(* HMI Lights Control *) //-----------------------------------------------------------------------------------------------
GVL_IO.gRelayOutputs.bSampleRecoveryLight 		:= GVL_HMI.bLightsToggleButton;
GVL_IO.gRelayOutputs.bStageCollectionLeftLight 	:= GVL_HMI.bLightsToggleButton;
GVL_IO.gRelayOutputs.bStageCollectionRightLight := GVL_HMI.bLightsToggleButton;

(* <Linear Pumps Old Position> ----------------------------------------------------------------------------------------- *)
// display linear pumps old position saved on persistent memory when in Calibration Mode
IF GVL_HMI.eMachineMode = E_MachineMode.CALIBRATION THEN
	FOR i := 1 TO 10 DO
		IF GVL_Motion.aPumps[i].Linear.iHomed THEN
			GVL_HMI.aCalibLinearPumps[1].rNewPosition := GVL_Motion.aPumps[i].Linear.rActualPos;
		END_IF
	END_FOR
END_IF

(* <Pump Factor Showing> ----------------------------------------------------------------------------------------------- *)
(*IF GVL_HMI.eMachineMode = E_MachineMode.CALIBRATION THEN
	FOR i := 1 TO 10 DO
		GVL_HMI.aCalPumpResults[i].rPumpFactor := GVL_Motion.aPumps[i].Rotary.rPumpFactorFromCalBox;
	END_FOR
END_IF
*)

(* <Safety Controls> ----------------------------------------------------------------------------------------------------*)
ton500ms(IN := NOT ton500ms.Q, PT := T#500MS);

IF ton500ms.Q THEN ACT_IOControls(); END_IF

//Calibration Box presence
GVL_HMI.bHMICalibrationBox := GVL_IO.gDigInputs.bCalibrationBoxPresent;

//Valves Angle
GVL_HMI.HMIAnimation.aValveAngle[1]	:= GVL_Motion.aValves[1].rActualPosition / 60;
GVL_HMI.HMIAnimation.aValveAngle[2]	:= GVL_Motion.aValves[2].rActualPosition / 60;;
GVL_HMI.HMIAnimation.aValveAngle[3]	:= GVL_Motion.aValves[3].rActualPosition / 60;;
GVL_HMI.HMIAnimation.aValveAngle[4]	:= GVL_Motion.aValves[4].rActualPosition / 60;;
GVL_HMI.HMIAnimation.aValveAngle[5]	:= GVL_Motion.aValves[5].rActualPosition / 60;;

//Pumps status Running or busy
IF GVL_HMI.eMachineMode = E_MachineMode.MANUAL THEN
	FOR i := 1 TO 10 DO
		aPumpStatus[i] := GVL_Motion.aPumpsRotary[i].GetStatus();
		GVL_HMI.aManualPumpsCmd[i].bBusy := NOT GVL_Motion.aPumps[i].Rotary.iNotMoving; //aPumpStatus[i].bBusy;
	END_FOR
END_IF

//Check if there is at least one pump running
GVL_Motion.bAnyPumpRunning := FALSE;
FOR i := 1 TO 10 DO
	IF GVL_HMI.aManualPumpsCmd[i].bBusy THEN
		GVL_Motion.bAnyPumpRunning := TRUE;
		EXIT;
	END_IF
END_FOR


//Pumps Animation | Calibration Screen
IF GVL_HMI.eMachineMode = E_MachineMode.CALIBRATION THEN
	ACT_CalibrationArrows();
END_IF

//Scan period for hmi refresh
//IF GVL_HMI.eMachineMode <> E_MachineMode.CALIBRATION AND GVL_HMI.eMachineMode <> E_MachineMode.MANUAL THEN
	fbHMIScan(bEnable := GVL_HMI.bHomeScreenLoaded, tPeriod := T#500MS);
	GVL_HMI.bMachineModeScan := fbHMIScan.bBlink;
//ELSE
//	GVL_HMI.bMachineModeScan := FALSE;
//END_IF

// Home Rotary Pumps direction cover
IF GVL_HMI.bHomeScreenLoaded THEN
	FOR i := 1 TO 10 DO
		GVL_HMI.HMIAnimation.bPumpPositiveDirection[i] := GVL_Motion.aPumps[i].Rotary.bPositiveDirection;
		GVL_HMI.HMIAnimation.bPumpNegativeDirection[i] := GVL_Motion.aPumps[i].Rotary.bNegativeDirection;
	END_FOR	
END_IF

//Doors hide/visible 
GVL_HMI.HMIAnimation.bHMIDoorOpen[1] := NOT GVL_Safety.SafetyInputs.bStageCollectLeftDoorFdbk;
GVL_HMI.HMIAnimation.bHMIDoorOpen[2] := NOT GVL_Safety.SafetyInputs.bStageCollectRightDoorFdbk;
GVL_HMI.HMIAnimation.bHMIDoorOpen[3] := NOT GVL_Safety.SafetyInputs.bSampleRecoveryDoorFdbk;
GVL_HMI.HMIAnimation.bHMIDoorOpen[4] := GVL_IO.gDigInputs.bAccessDoor4InterlockFdbk;
GVL_HMI.HMIAnimation.bHMIDoorOpen[5] := GVL_IO.gDigInputs.bAccessDoor5InterlockFdbk;
GVL_HMI.HMIAnimation.bHMIDoorOpen[6] := GVL_IO.gDigInputs.bAccessDoor6InterlockFdbk;

//Doors open blinking red alert
fbBlinkDoor[1](bEnable := NOT GVL_Safety.SafetyInputs.bStageCollectLeftDoorFdbk, tPeriod := T#1S);
GVL_HMI.HMIAnimation.bHMIDoorBlink[1] := fbBlinkDoor[1].bBlink;

fbBlinkDoor[2](bEnable := NOT GVL_Safety.SafetyInputs.bStageCollectRightDoorFdbk, tPeriod := T#1S);
GVL_HMI.HMIAnimation.bHMIDoorBlink[2] := fbBlinkDoor[2].bBlink;

fbBlinkDoor[3](bEnable := NOT GVL_Safety.SafetyInputs.bSampleRecoveryDoorFdbk, tPeriod := T#1S);
GVL_HMI.HMIAnimation.bHMIDoorBlink[3] := fbBlinkDoor[3].bBlink;

fbBlinkDoor[4](bEnable := GVL_IO.gDigInputs.bAccessDoor4InterlockFdbk, tPeriod := T#1S);
GVL_HMI.HMIAnimation.bHMIDoorBlink[4] := fbBlinkDoor[4].bBlink;

fbBlinkDoor[5](bEnable := GVL_IO.gDigInputs.bAccessDoor5InterlockFdbk, tPeriod := T#1S);
GVL_HMI.HMIAnimation.bHMIDoorBlink[5] := fbBlinkDoor[5].bBlink;

fbBlinkDoor[6](bEnable := GVL_IO.gDigInputs.bAccessDoor6InterlockFdbk, tPeriod := T#1S);
GVL_HMI.HMIAnimation.bHMIDoorBlink[6] := fbBlinkDoor[6].bBlink;


(* <\Controls Animation> *********************************************************************************************** *)

(* <Icons Animation> *************************************************************************************************** *)
IF NOT bFirstIconSet THEN
	GVL_HMI.HMIAnimation.eIconStateSafety   := E_IconState.Waiting;
	GVL_HMI.HMIAnimation.eIconStateAirFlow  := E_IconState.Waiting;
	GVL_HMI.HMIAnimation.eIconStateSealing 	:= E_IconState.Waiting;
	GVL_HMI.HMIAnimation.eIconStateHardware := E_IconState.Waiting;
	GVL_HMI.HMIAnimation.eIconStatePrime 	:= E_IconState.Waiting;
	GVL_HMI.HMIAnimation.eIconStateLeakTest := E_IconState.Waiting;
	GVL_HMI.HMIAnimation.eIconStateRecovery := E_IconState.Waiting;
	GVL_HMI.HMIAnimation.eIconStateWashing  := E_IconState.Waiting;
	GVL_HMI.HMIAnimation.eIconStateDry 		:= E_IconState.Waiting;
	bFirstIconSet := TRUE;
END_IF

IF GVL_HMI.eMachineMode = E_MachineMode.IMEDIATE_FAULT THEN
	GVL_HMI.HMIAnimation.eIconStateSafety   := E_IconState.Waiting;
	GVL_HMI.HMIAnimation.eIconStateAirFlow  := E_IconState.Waiting;
	GVL_HMI.HMIAnimation.eIconStateSealing  := E_IconState.Waiting;
	GVL_HMI.HMIAnimation.eIconStateHardware := E_IconState.Waiting;
	GVL_HMI.HMIAnimation.eIconStatePrime  	:= E_IconState.Waiting;
	GVL_HMI.HMIAnimation.eIconStateLeakTest := E_IconState.Waiting;
	GVL_HMI.HMIAnimation.eIconStateRecovery := E_IconState.Waiting;
	GVL_HMI.HMIAnimation.eIconStateWashing  := E_IconState.Waiting;
	GVL_HMI.HMIAnimation.eIconStateDry 	    := E_IconState.Waiting;
ELSE
	GVL_HMI.HMIAnimation.eIconStateSafety := E_IconState.Completed;
END_IF

IF GVL_HMI.eMachineMode = E_MachineMode.STOPPED THEN
	GVL_HMI.HMIAnimation.eIconStateSafety   := E_IconState.Waiting;
	GVL_HMI.HMIAnimation.eIconStateAirFlow  := E_IconState.Waiting;
	GVL_HMI.HMIAnimation.eIconStateSealing 	:= E_IconState.Waiting;
	GVL_HMI.HMIAnimation.eIconStateHardware := E_IconState.Waiting;
	GVL_HMI.HMIAnimation.eIconStatePrime 	:= E_IconState.Waiting;
	GVL_HMI.HMIAnimation.eIconStateLeakTest := E_IconState.Waiting;
	GVL_HMI.HMIAnimation.eIconStateRecovery := E_IconState.Waiting;
	GVL_HMI.HMIAnimation.eIconStateWashing  := E_IconState.Waiting;
	GVL_HMI.HMIAnimation.eIconStateDry 	    := E_IconState.Waiting;
END_IF

(* <\Icons Animation> *************************************************************************************************** *)

(* <Machine Settings> ************************************************************************************************** *)
IF GVL_HMI.bSaveParametersBt THEN // Save Settings button from HMI
	GVL_Settings.stMachineParam	 		:= GVL_HMI.HMIParameters; 		 // Motion Settings
	GVL_Settings.stCalibParameters 		:= GVL_HMI.stHMICalibParameters; // Calibration Settings
	GVL_Settings.stPumpParameters 		:= GVL_HMI.stHMIPumpParameters;	 // Pump Settings
	GVL_Settings.stLeakTestParameters 	:= GVL_HMI.stLeakTestParameters; // Leak Test Settings
	GVL_Settings.sLastSysSettingsChangedBy 	:= GVL_HMI.sUserNameEventTriggered;
	GVL_Settings.sLastSysSettingsChangedOn 	:= GVL_HMI.sDateAndTimeEventTriggered;
	GVL_Settings.sysRevNumber 				:= GVL_Settings.sysRevNumber + 1;
	DB_Query.state:= E_DB_QUERY_STATE.INSERT_SYS_PARAMETERS;	// DB writing
	GVL_HMI.bSaveParametersBt 	:= FALSE;
	GVL_HMI.bSaveParametersDone := TRUE;
END_IF

IF GVL_HMI.bReloadHMIParameters OR (GVL_HMI.eMachineMode = E_MachineMode.CALIBRATION) THEN
	GVL_HMI.HMIParameters := GVL_Settings.stMachineParam;				 // Motion Settings
	GVL_HMI.stHMICalibParameters := GVL_Settings.stCalibParameters; 	 // Calibration Settings
	GVL_HMI.stHMIPumpParameters  := GVL_Settings.stPumpParameters; 		 // Pump Settings
	GVL_HMI.stLeakTestParameters := GVL_Settings.stLeakTestParameters; 	 // Leak Test Settings
	GVL_HMI.bReloadHMIParameters := FALSE;
END_IF

// Solvents Section [Database insert done via HMI]
PRG_SaveSolvents();
(*
IF GVL_HMI.bSaveSolventsBt THEN
	GVL_Settings.stSolventsInfo := GVL_HMI.stHMISolventsInfo;	// Solvents info snapshot
	GVL_HMI.bSaveSolventsBt := FALSE;
END_IF
*)
(* <\Machine Settings> ************************************************************************************************** *)

(* <HMI Alerts> ********************************************************************************************************* *)

//Auto Cycle Incoherence [when there is something missing to start the auto cycle] 
GVL_HMI.bIncoherenceDetected := (NOT GVL_Recipe.bIsThereRecipeActivated) OR (NOT GVL_IO.gDigInputs.bThroatJigPresent) OR (NOT GVL_IO.bVialRackPresent) OR bSolventIssue OR GVL_IO.gDigInputs.bWasteOverflowSensor;

bSolventIssue := GVL_Alarms.aSolventLowLevel[1] OR GVL_Alarms.aSolventLowLevel[2] OR GVL_Alarms.aSolventLowLevel[3] OR GVL_Alarms.aSolventLowLevel[4] OR GVL_Alarms.bWasteHighLevel;

IF GVL_HMI.HMIAnimation.rWasteLevel	> 70 THEN
	GVL_Alarms.bWasteHighLevel := TRUE;
ELSE
	GVL_Alarms.bWasteHighLevel := FALSE;
END_IF

IF GVL_Recipe.bIsThereRecipeActivated THEN
	//Checking solvent levels of Rinse 1 Solvent
	CASE GVL_Recipe.stActiveRecipe.stSolventsTimes.aSolventN[1] OF
	1:
		IF GVL_HMI.HMIAnimation.aSolventLevel[1] < 30 THEN
			GVL_Alarms.aSolventLowLevel[1] := TRUE;
		ELSE
			GVL_Alarms.aSolventLowLevel[1] := FALSE;
		END_IF
	2:
		IF GVL_HMI.HMIAnimation.aSolventLevel[2] < 30 THEN
			GVL_Alarms.aSolventLowLevel[2] := TRUE;
		ELSE
			GVL_Alarms.aSolventLowLevel[2] := FALSE;
		END_IF

	3:
		IF GVL_HMI.HMIAnimation.aSolventLevel[3] < 30 THEN
			GVL_Alarms.aSolventLowLevel[3] := TRUE;
		ELSE
			GVL_Alarms.aSolventLowLevel[3] := FALSE;
		END_IF
	4:
		IF GVL_HMI.HMIAnimation.aSolventLevel[4] < 30 THEN
			GVL_Alarms.aSolventLowLevel[4] := TRUE;
		ELSE
			GVL_Alarms.aSolventLowLevel[4] := FALSE;
		END_IF
	END_CASE 
	
	//Checking solvent levels of Rinse 2 Solvent
	CASE GVL_Recipe.stActiveRecipe.stSolventsTimes.aSolventN[2] OF
	1:
		IF GVL_HMI.HMIAnimation.aSolventLevel[1] < 30 THEN
			GVL_Alarms.aSolventLowLevel[1] := TRUE;
		ELSE
			GVL_Alarms.aSolventLowLevel[1] := FALSE;
		END_IF
	2:
		IF GVL_HMI.HMIAnimation.aSolventLevel[2] < 30 THEN
			GVL_Alarms.aSolventLowLevel[2] := TRUE;
		ELSE
			GVL_Alarms.aSolventLowLevel[2] := FALSE;
		END_IF

	3:
		IF GVL_HMI.HMIAnimation.aSolventLevel[3] < 30 THEN
			GVL_Alarms.aSolventLowLevel[3] := TRUE;
		ELSE
			GVL_Alarms.aSolventLowLevel[3] := FALSE;
		END_IF
	4:
		IF GVL_HMI.HMIAnimation.aSolventLevel[4] < 30 THEN
			GVL_Alarms.aSolventLowLevel[4] := TRUE;
		ELSE
			GVL_Alarms.aSolventLowLevel[4] := FALSE;
		END_IF
	END_CASE 
END_IF

//-------------------------------------------------

IF GVL_Recipe.bIsThereRecipeActivated THEN
	GVL_HMI.sActivatedRecipeHomeNaming := concat(GVL_Recipe.stActiveRecipe.stInfo.sMethodName,concat(' | Created by ', concat(GVL_Recipe.stActiveRecipe.stInfo.sCreatedBy,concat(' on ', DATE_TO_STRING(GVL_Recipe.stActiveRecipe.stInfo.dCreationDate)))));
ELSE
	GVL_HMI.sActivatedRecipeHomeNaming := 'There is no Recipe Activated';
END_IF

(* <\HMI Alerts> ******************************************************************************************************* *)
(* Motors Interlock *) // Releasing alarm trigger after 2 seconds.
IF GVL_HMI.bM1MoveNotAllowedTrigger THEN
	tonInterlockReleaseM1(In := TRUE, PT := T#2S);
ELSE
	tonInterlockReleaseM1(In := FALSE, PT := T#2S);
END_IF

IF GVL_HMI.bM2MoveNotAllowedTrigger THEN
	tonInterlockReleaseM2(In := TRUE, PT := T#2S);
ELSE
	tonInterlockReleaseM2(In := FALSE, PT := T#2S);
END_IF

IF GVL_HMI.bM3MoveNotAllowedTrigger THEN
	tonInterlockReleaseM3(In := TRUE, PT := T#2S);
ELSE
	tonInterlockReleaseM3(In := FALSE, PT := T#2S);
END_IF

IF tonInterlockReleaseM1.Q THEN
	GVL_HMI.bM1MoveNotAllowedTrigger := FALSE;
END_IF

IF tonInterlockReleaseM2.Q THEN
	GVL_HMI.bM2MoveNotAllowedTrigger := FALSE;
END_IF

IF tonInterlockReleaseM3.Q THEN
	GVL_HMI.bM3MoveNotAllowedTrigger := FALSE;
END_IF

(* <HMI Report Listing> ******************************************************************************************************* *)



(* <\HMI Report Listing> ******************************************************************************************************* *)

(* <HMI Reminders> ******************************************************************************************************* *)

GVL_HMI.stReminders.bRecipeActivated 	:= GVL_Recipe.bIsThereRecipeActivated;
//GVL_HMI.stReminders.bSolventLevels 		:= GVL_Recipe.bIsThereRecipeActivated OR GVL_Alarms.aSolventLowLevel[1] OR GVL_Alarms.aSolventLowLevel[2] OR GVL_Alarms.aSolventLowLevel[3] OR GVL_Alarms.aSolventLowLevel[4]; // TODO - only evaluate the levels used on recipe
GVL_HMI.stReminders.bWasteLevel 		:= GVL_Alarms.bWasteHighLevel;
GVL_HMI.stReminders.bThroatJigPresent	:= GVL_IO.gDigInputs.bThroatJigPresent;
GVL_HMI.stReminders.bVialRackPresent	:= GVL_IO.bVialRackPresent;
GVL_HMI.stReminders.bVialRackRemoved	:= NOT GVL_IO.bVialRackPresent;
GVL_HMI.stReminders.bCalBoxInPlace		:= GVL_IO.gDigInputs.bCalibrationBoxPresent;
GVL_HMI.stReminders.bStagePlateHomePos	:= (GVL_Motion.M1Motor.rActualPos > -10 AND GVL_Motion.M1Motor.rActualPos < 10);

GVL_HMI.stReminders.bSolventLevels :=
    GVL_Recipe.bIsThereRecipeActivated
    AND
    (
        (GVL_Recipe.stActiveRecipe.stSolventsTimes.aSolventN[1] = 0
         OR_ELSE NOT GVL_Alarms.aSolventLowLevel[GVL_Recipe.stActiveRecipe.stSolventsTimes.aSolventN[1]])
    )
    AND
    (
        (GVL_Recipe.stActiveRecipe.stSolventsTimes.aSolventN[2] = 0
         OR_ELSE NOT GVL_Alarms.aSolventLowLevel[GVL_Recipe.stActiveRecipe.stSolventsTimes.aSolventN[2]])
    )
    AND
    (
        (GVL_Recipe.stActiveRecipe.stSolventsTimes.aSolventN[3] = 0
         OR_ELSE NOT GVL_Alarms.aSolventLowLevel[GVL_Recipe.stActiveRecipe.stSolventsTimes.aSolventN[3]])
    )
    AND
    (
        (GVL_Recipe.stActiveRecipe.stSolventsTimes.aSolventN[4] = 0
         OR_ELSE NOT GVL_Alarms.aSolventLowLevel[GVL_Recipe.stActiveRecipe.stSolventsTimes.aSolventN[4]])
    );


GVL_HMI.stReminders.bAutoCicleReady		:= GVL_HMI.stReminders.bRecipeActivated AND GVL_HMI.stReminders.bSolventLevels AND GVL_HMI.stReminders.bWasteLevel  AND GVL_HMI.stReminders.bThroatJigPresent AND GVL_HMI.stReminders.bVialRackPresent;
GVL_HMI.stReminders.bCalibrationReady	:= GVL_HMI.stReminders.bVialRackRemoved AND GVL_HMI.stReminders.bCalBoxInPlace AND GVL_HMI.stReminders.bStagePlateHomePos;


(* <\HMI Reminders> ******************************************************************************************************* *)

(* <TEMP ******************************************************************************************************* *)
IF GVL_HMI.bResetM1MotorBt THEN
	GVL_HMI.bResetM1MotorBt := NOT GVL_Motion.aMotors[1].Reset();
END_IF

ACTION ACT_CalibrationArrows:
(* Pumps arrow animation *)
//Get pump Status
FOR i := 1 TO 10 DO
	aPumpStatus[i] := GVL_Motion.aPumpsRotary[i].GetStatus();
END_FOR

//Blink aPumpMovingFwd[i] if moving forward
FOR i := 1 TO 10 DO
	fbBlinkPumpArrowFWD[i]( bEnable := aPumpStatus[i].bMovingFwd, tPeriod := T#500MS );
	GVL_HMI.HMIAnimation.aPumpingArrowFwd[i] := fbBlinkPumpArrowFWD[i].bBlink;
END_FOR

//Blink aPumpMovingBwd[i] if moving backwards
FOR i := 1 TO 10 DO
	fbBlinkPumpArrowBWD[i]( bEnable := aPumpStatus[i].bMovingBck, tPeriod := T#500MS );
	GVL_HMI.HMIAnimation.aPumpingArrowBwd[i] := fbBlinkPumpArrowBWD[i].bBlink;
END_FOR
END_ACTION

ACTION ACT_IOControls:

(* <EL6910 Terminal 3> -------------------------------------------------------------------------------------------------------------*)
GVL_IO.stEL6910.qSafetyRun 			:= GVL_Safety.bSafetyRun;
GVL_IO.stEL6910.qSafetyErrorAck 	:= GVL_Safety.bSafetyErrorAck;
GVL_IO.stEL6910.qSafetyAirPresureOK := GVL_Safety.SafetyOutputs.bAirPressureOK;
GVL_IO.stEL6910.iSafetyOK 			:= GVL_Safety.bSafetyEnable;
GVL_IO.stEL6910.qLockDoorsCommand	:= GVL_Safety.bDoorLockCommand;
GVL_IO.stEL6910.iBypassDoor3Command := GVL_Safety.bDoor3BypassAccepted;


(* <EL1918 Terminal 4> -------------------------------------------------------------------------------------------------------------*)
GVL_HMI.aIOTerm04[1] := GVL_Safety.SafetyInputs.bEStopHMICh1;
GVL_HMI.aIOTerm04[2] := GVL_Safety.SafetyInputs.bEStopHMICh2;
GVL_HMI.aIOTerm04[3] := GVL_Safety.SafetyInputs.bEStopSideCh1;
GVL_HMI.aIOTerm04[4] := GVL_Safety.SafetyInputs.bEStopSideCh2;
GVL_HMI.aIOTerm04[5] := GVL_Safety.SafetyInputs.bMachineReset;
GVL_HMI.aIOTerm04[6] := GVL_Safety.SafetyInputs.bStageCollectLeftDoorCh1;
GVL_HMI.aIOTerm04[7] := GVL_Safety.SafetyInputs.bStageCollectLeftDoorCh2;
GVL_HMI.aIOTerm04[8] := GVL_Safety.SafetyInputs.bStageCollectLeftDoorFdbk;

(* <EL1918 Terminal 5> -------------------------------------------------------------------------------------------------------------*)
GVL_HMI.aIOTerm05[1] := GVL_Safety.SafetyInputs.bStageCollectRightDoorCh1;
GVL_HMI.aIOTerm05[2] := GVL_Safety.SafetyInputs.bStageCollectRightDoorCh2;
GVL_HMI.aIOTerm05[3] := GVL_Safety.SafetyInputs.bStageCollectRightDoorFdbk;
GVL_HMI.aIOTerm05[4] := GVL_Safety.SafetyInputs.bSampleRecoveryDoorCh1;
GVL_HMI.aIOTerm05[5] := GVL_Safety.SafetyInputs.bSampleRecoveryDoorCh2;
GVL_HMI.aIOTerm05[6] := GVL_Safety.SafetyInputs.bSampleRecoveryDoorFdbk;
GVL_HMI.aIOTerm05[7] := FALSE;
GVL_HMI.aIOTerm05[8] := FALSE;

(* <EL1918 Terminal 6> -------------------------------------------------------------------------------------------------------------*)
GVL_HMI.aIOTerm06[1] := NOT GVL_Safety.SafetyInputs.bFestoMS6ValveFdbk;
GVL_HMI.aIOTerm06[2] := GVL_Safety.SafetyInputs.bFestoMS6DumpValveFdbk;
GVL_HMI.aIOTerm06[3] := NOT GVL_Safety.SafetyInputs.bD4AccessDoorIntlckOSSD1;
GVL_HMI.aIOTerm06[4] := NOT GVL_Safety.SafetyInputs.bD4AccessDoorIntlckOSSD2;
GVL_HMI.aIOTerm06[5] := NOT GVL_Safety.SafetyInputs.bD5AccessDoorIntlckOSSD1;
GVL_HMI.aIOTerm06[6] := NOT GVL_Safety.SafetyInputs.bD5AccessDoorIntlckOSSD2;
GVL_HMI.aIOTerm06[7] := NOT GVL_Safety.SafetyInputs.bD6AccessDoorIntlckOSSD1;
GVL_HMI.aIOTerm06[8] := NOT GVL_Safety.SafetyInputs.bD6AccessDoorIntlckOSSD2;

(* <EL2904 Terminal 7> -------------------------------------------------------------------------------------------------------------*)
GVL_HMI.aIOTerm07[1] := GVL_Safety.aEL2904_T07[1];
GVL_HMI.aIOTerm07[2] := GVL_Safety.aEL2904_T07[2];
GVL_HMI.aIOTerm07[3] := GVL_Safety.aEL2904_T07[3];
GVL_HMI.aIOTerm07[4] := GVL_Safety.aEL2904_T07[4];

(* <EL2904 Terminal 8> -------------------------------------------------------------------------------------------------------------*)
GVL_HMI.aIOTerm08[1] := GVL_Safety.aEL2904_T08[1];
GVL_HMI.aIOTerm08[2] := GVL_Safety.aEL2904_T08[2];
GVL_HMI.aIOTerm08[3] := GVL_Safety.aEL2904_T08[3];
GVL_HMI.aIOTerm08[4] := GVL_Safety.aEL2904_T08[4];

(* <EL1809 Terminal 9> -------------------------------------------------------------------------------------------------------------*)
GVL_HMI.aIOTerm09[1] := GVL_IO.gDigInputs.bStartButton;
GVL_HMI.aIOTerm09[2] := GVL_IO.gDigInputs.bStopButton;
GVL_HMI.aIOTerm09[3] := GVL_IO.gDigInputs.b24VPowerSupplyOK;
GVL_HMI.aIOTerm09[4] := GVL_IO.gDigInputs.b24VPowerSupplyOKBck;
GVL_HMI.aIOTerm09[5] := GVL_IO.gDigInputs.b48VPowerSupplyOK;
GVL_HMI.aIOTerm09[6] := GVL_IO.gDigInputs.bStageCollection_Home;
GVL_HMI.aIOTerm09[7] := GVL_IO.gDigInputs.bSampleRecovery_Vertical_Home;
GVL_HMI.aIOTerm09[8] := GVL_IO.gDigInputs.bSampleRecovery_Horizontal_Home;
GVL_HMI.aIOTerm09[9] := GVL_IO.gDigInputs.bWasteOverflowSensor;
GVL_HMI.aIOTerm09[10] := GVL_IO.gDigInputs.bUPSReady;
GVL_HMI.aIOTerm09[11] := GVL_IO.gDigInputs.bUPSReplaceBattery;
GVL_HMI.aIOTerm09[12] := GVL_IO.gDigInputs.b48VPowerSupplyOKBck;
GVL_HMI.aIOTerm09[13] := GVL_IO.gDigInputs.bCalibrationBoxPresent;
GVL_HMI.aIOTerm09[14] := GVL_IO.gDigInputs.bThroatJigPresent;
GVL_HMI.aIOTerm09[15] := FALSE;
GVL_HMI.aIOTerm09[16] := FALSE;

(* <EL2809 Terminal 10> -------------------------------------------------------------------------------------------------------------*)
GVL_HMI.aIOTerm10[1] := GVL_IO.gDigOutputs.bStartIndicator;
GVL_HMI.aIOTerm10[2] := GVL_IO.gDigOutputs.bResetIndicator;
GVL_HMI.aIOTerm10[3] := GVL_IO.gDigOutputs.bTowerRedLight;
GVL_HMI.aIOTerm10[4] := GVL_IO.gDigOutputs.bTowerAmberLight;
GVL_HMI.aIOTerm10[5] := GVL_IO.gDigOutputs.bTowerGreenLight;
GVL_HMI.aIOTerm10[6] := GVL_IO.gDigOutputs.bTowerBuzzer;
GVL_HMI.aIOTerm10[7] := GVL_IO.gDigOutputs.bSolenoidValveB;
GVL_HMI.aIOTerm10[8] := GVL_IO.gDigOutputs.bSolenoidValveA;
GVL_HMI.aIOTerm10[9] := GVL_IO.gDigOutputs.bSolenoidValveC;
GVL_HMI.aIOTerm10[10] := FALSE;
GVL_HMI.aIOTerm10[11] := FALSE;
GVL_HMI.aIOTerm10[12] := FALSE;
GVL_HMI.aIOTerm10[13] := FALSE;
GVL_HMI.aIOTerm10[14] := FALSE;
GVL_HMI.aIOTerm10[15] := FALSE;
GVL_HMI.aIOTerm10[16] := FALSE;

(* <EL2624 Terminal 11> -------------------------------------------------------------------------------------------------------------*)
GVL_HMI.aIOTerm11[1] := GVL_IO.gRelayOutputs.bStageCollectionLeftLight;
GVL_HMI.aIOTerm11[2] := GVL_IO.gRelayOutputs.bSampleRecoveryLight;
GVL_HMI.aIOTerm11[3] := GVL_IO.gRelayOutputs.bStageCollectionRightLight;
GVL_HMI.aIOTerm11[4] := FALSE;

(* <EL9410 Terminal 12> -------------------------------------------------------------------------------------------------------------*)
GVL_HMI.aIOTerm12[1] := GVL_IO.bEL9410UPStatus;
GVL_HMI.aIOTerm12[2] := GVL_IO.bEL9410USStatus;

(* <EL3058 Terminal 13> -------------------------------------------------------------------------------------------------------------*)
GVL_HMI.aIOTerm13[1] := GVL_IO.gAnalogInputs.rMainPressureSupplyInput;
GVL_HMI.aIOTerm13[2] := GVL_IO.gAnalogInputs.rLeakTestPressureSensor;
GVL_HMI.aIOTerm13[3] := GVL_IO.gAnalogInputs.rPressureRegulatorInput;
GVL_HMI.aIOTerm13[3] := 0.0;

(* <EL9576 Terminal 14> -------------------------------------------------------------------------------------------------------------*)
GVL_HMI.aIOTerm14[1] := GVL_IO.bEL9576T14Overtemp;
GVL_HMI.aIOTerm14[2] := GVL_IO.bEL9576T14I2TError;
GVL_HMI.aIOTerm14[3] := GVL_IO.bEL9576T14I2TWarning;
GVL_HMI.aIOTerm14[4] := GVL_IO.bEL9576T14OverVoltage;
GVL_HMI.aIOTerm14[5] := GVL_IO.bEL9576T14UnderVoltage;
GVL_HMI.aIOTerm14[6] := GVL_IO.bEL9576T14ChopperOn;
GVL_HMI.aIOTerm14[7] := GVL_IO.bEL9576T14OverCurrent;
GVL_HMI.iIOTerm14DCIn := GVL_IO.bEL9576T14DCLinkVoltage;

(* <EL7211 Terminal 15> -------------------------------------------------------------------------------------------------------------*)
GVL_HMI.aIOTerm15[1] := GVL_Motion.M2Motor.iOperational;
GVL_HMI.aIOTerm15[2] := GVL_Motion.M2Motor.iHomed;
GVL_HMI.aIOTerm15[3] := GVL_Motion.M2Motor.iError;
GVL_HMI.aIOTerm15Values[1] := LINT_TO_LREAL(TRUNC(GVL_Motion.M2Motor.rActualPosition*1000)) / 1000.0;
GVL_HMI.aIOTerm15Values[2] := LINT_TO_LREAL(TRUNC(GVL_Motion.M2Motor.rActualVel*1000)) / 1000.0;
GVL_HMI.aIOTerm15Values[3] := LINT_TO_LREAL(TRUNC(GVL_Motion.M2Motor.rActualTorque*1000)) / 1000.0;
GVL_HMI.iIOTerm15ErrorCode := GVL_Motion.M2Motor.nErrorCode;

(* <EL7211 Terminal 16> -------------------------------------------------------------------------------------------------------------*)
GVL_HMI.aIOTerm16[1] := GVL_Motion.M3Motor.iOperational;
GVL_HMI.aIOTerm16[2] := GVL_Motion.M3Motor.iHomed;
GVL_HMI.aIOTerm16[3] := GVL_Motion.M3Motor.iError;
GVL_HMI.aIOTerm16Values[1] := LINT_TO_LREAL(TRUNC(GVL_Motion.M3Motor.rActualPosition*1000)) / 1000.0;
GVL_HMI.aIOTerm16Values[2] := LINT_TO_LREAL(TRUNC(GVL_Motion.M3Motor.rActualVel*1000)) / 1000.0;
GVL_HMI.aIOTerm16Values[3] := LINT_TO_LREAL(TRUNC(GVL_Motion.M3Motor.rActualTorque*1000)) / 1000.0;
GVL_HMI.iIOTerm16ErrorCode := GVL_Motion.M3Motor.nErrorCode;

(* <EL3022 Terminal 17> -------------------------------------------------------------------------------------------------------------*)
GVL_HMI.aIOTerm17[1] := GVL_IO.bEL3022ChAUnderRange;
GVL_HMI.aIOTerm17[2] := GVL_IO.bEL3022ChAOverRange;
GVL_HMI.aIOTerm17[3] := GVL_IO.bEL3022ChAError;
GVL_HMI.aIOTerm17[4] := GVL_IO.bEL3022ChBUnderRange;
GVL_HMI.aIOTerm17[5] := GVL_IO.bEL3022ChBOverRange;
GVL_HMI.aIOTerm17[6] := GVL_IO.bEL3022ChBError;
GVL_HMI.aIOTerm17Values[1] := 0.0;
GVL_HMI.aIOTerm17Values[2] := 0.0;

(* <EL1809 Terminal 18> -------------------------------------------------------------------------------------------------------------*)
GVL_HMI.aIOTerm18[1] := NOT GVL_IO.gDigInputs.bAccessDoor4InterlockFdbk;
GVL_HMI.aIOTerm18[2] := NOT GVL_IO.gDigInputs.bAccessDoor5InterlockFdbk;
GVL_HMI.aIOTerm18[3] := NOT GVL_IO.gDigInputs.bAccessDoor6InterlockFdbk;
GVL_HMI.aIOTerm18[4] := FALSE;
GVL_HMI.aIOTerm18[5] := FALSE;
GVL_HMI.aIOTerm18[6] := FALSE;
GVL_HMI.aIOTerm18[7] := FALSE;
GVL_HMI.aIOTerm18[8] := FALSE;
GVL_HMI.aIOTerm18[9] := FALSE;
GVL_HMI.aIOTerm18[10] := FALSE;
GVL_HMI.aIOTerm18[11] := FALSE;
GVL_HMI.aIOTerm18[12] := FALSE;
GVL_HMI.aIOTerm18[13] := FALSE;
GVL_HMI.aIOTerm18[14] := FALSE;
GVL_HMI.aIOTerm18[15] := FALSE;
GVL_HMI.aIOTerm18[16] := FALSE;

(* <EL2904 Terminal 19> -------------------------------------------------------------------------------------------------------------*)
GVL_HMI.aIOTerm19[1] := GVL_Safety.aEL2904_T19[1];
GVL_HMI.aIOTerm19[2] := GVL_Safety.aEL2904_T19[2];
GVL_HMI.aIOTerm19[3] := GVL_Safety.aEL2904_T19[3];
GVL_HMI.aIOTerm19[4] := GVL_Safety.aEL2904_T19[4];

(* <EL7062 Terminal 23> -------------------------------------------------------------------------------------------------------------*)
GVL_HMI.stIOTerm23.bAxisOperational[1] 	:= GVL_Motion.aPumps[1].Linear.iOperational;
GVL_HMI.stIOTerm23.rActualPosition[1] 	:= GVL_Motion.aPumps[1].Linear.rActualPos;
GVL_HMI.stIOTerm23.rActualVelocity[1] 	:= GVL_Motion.aPumps[1].Linear.rActualVel;
GVL_HMI.stIOTerm23.rActualTorque[1] 	:= GVL_Motion.aPumps[1].Linear.rActualTorque;
GVL_HMI.stIOTerm23.bAxisHomed[1] 		:= GVL_Motion.aPumps[1].Linear.iHomed;
GVL_HMI.stIOTerm23.bAxisError[1] 		:= GVL_Motion.aPumps[1].Linear.iError;
GVL_HMI.stIOTerm23.nErrorCode[1] 		:= GVL_Motion.aPumps[1].Linear.nErrorCode;
GVL_HMI.stIOTerm23.bAxisOperational[2] 	:= GVL_Motion.aPumps[1].Rotary.iOperational;
GVL_HMI.stIOTerm23.rActualPosition[2] 	:= GVL_Motion.aPumps[1].Rotary.rActualPos;
GVL_HMI.stIOTerm23.rActualVelocity[2] 	:= GVL_Motion.aPumps[1].Rotary.rActualVel;
GVL_HMI.stIOTerm23.rActualTorque[2] 	:= GVL_Motion.aPumps[1].Rotary.rActualTorque;
GVL_HMI.stIOTerm23.bAxisHomed[2] 		:= GVL_Motion.aPumps[1].Rotary.iHomed;
GVL_HMI.stIOTerm23.bAxisError[2] 		:= GVL_Motion.aPumps[1].Rotary.iError;
GVL_HMI.stIOTerm23.nErrorCode[2] 		:= GVL_Motion.aPumps[1].Rotary.nErrorCode;

(* <EL7062 Terminal 24> -------------------------------------------------------------------------------------------------------------*)
GVL_HMI.stIOTerm24.bAxisOperational[1] 	:= GVL_Motion.aPumps[2].Linear.iOperational;
GVL_HMI.stIOTerm24.rActualPosition[1] 	:= GVL_Motion.aPumps[2].Linear.rActualPos;
GVL_HMI.stIOTerm24.rActualVelocity[1] 	:= GVL_Motion.aPumps[2].Linear.rActualVel;
GVL_HMI.stIOTerm24.rActualTorque[1] 	:= GVL_Motion.aPumps[2].Linear.rActualTorque;
GVL_HMI.stIOTerm24.bAxisHomed[1] 		:= GVL_Motion.aPumps[2].Linear.iHomed;
GVL_HMI.stIOTerm24.bAxisError[1] 		:= GVL_Motion.aPumps[2].Linear.iError;
GVL_HMI.stIOTerm24.nErrorCode[1] 		:= GVL_Motion.aPumps[2].Linear.nErrorCode;
GVL_HMI.stIOTerm24.bAxisOperational[2] 	:= GVL_Motion.aPumps[2].Rotary.iOperational;
GVL_HMI.stIOTerm24.rActualPosition[2] 	:= GVL_Motion.aPumps[2].Rotary.rActualPos;
GVL_HMI.stIOTerm24.rActualVelocity[2] 	:= GVL_Motion.aPumps[2].Rotary.rActualVel;
GVL_HMI.stIOTerm24.rActualTorque[2] 	:= GVL_Motion.aPumps[2].Rotary.rActualTorque;
GVL_HMI.stIOTerm24.bAxisHomed[2] 		:= GVL_Motion.aPumps[2].Rotary.iHomed;
GVL_HMI.stIOTerm24.bAxisError[2] 		:= GVL_Motion.aPumps[2].Rotary.iError;
GVL_HMI.stIOTerm24.nErrorCode[2] 		:= GVL_Motion.aPumps[2].Rotary.nErrorCode;

(* <EL7062 Terminal 25> -------------------------------------------------------------------------------------------------------------*)
GVL_HMI.stIOTerm25.bAxisOperational[1] 	:= GVL_Motion.aPumps[3].Linear.iOperational;
GVL_HMI.stIOTerm25.rActualPosition[1] 	:= GVL_Motion.aPumps[3].Linear.rActualPos;
GVL_HMI.stIOTerm25.rActualVelocity[1] 	:= GVL_Motion.aPumps[3].Linear.rActualVel;
GVL_HMI.stIOTerm25.rActualTorque[1] 	:= GVL_Motion.aPumps[3].Linear.rActualTorque;
GVL_HMI.stIOTerm25.bAxisHomed[1] 		:= GVL_Motion.aPumps[3].Linear.iHomed;
GVL_HMI.stIOTerm25.bAxisError[1] 		:= GVL_Motion.aPumps[3].Linear.iError;
GVL_HMI.stIOTerm25.nErrorCode[1] 		:= GVL_Motion.aPumps[3].Linear.nErrorCode;
GVL_HMI.stIOTerm25.bAxisOperational[2] 	:= GVL_Motion.aPumps[3].Rotary.iOperational;
GVL_HMI.stIOTerm25.rActualPosition[2] 	:= GVL_Motion.aPumps[3].Rotary.rActualPos;
GVL_HMI.stIOTerm25.rActualVelocity[2] 	:= GVL_Motion.aPumps[3].Rotary.rActualVel;
GVL_HMI.stIOTerm25.rActualTorque[2] 	:= GVL_Motion.aPumps[3].Rotary.rActualTorque;
GVL_HMI.stIOTerm25.bAxisHomed[2] 		:= GVL_Motion.aPumps[3].Rotary.iHomed;
GVL_HMI.stIOTerm25.bAxisError[2] 		:= GVL_Motion.aPumps[3].Rotary.iError;
GVL_HMI.stIOTerm25.nErrorCode[2] 		:= GVL_Motion.aPumps[3].Rotary.nErrorCode;

(* <EL7062 Terminal 26> -------------------------------------------------------------------------------------------------------------*)
GVL_HMI.stIOTerm26.bAxisOperational[1] 	:= GVL_Motion.aPumps[4].Linear.iOperational;
GVL_HMI.stIOTerm26.rActualPosition[1] 	:= GVL_Motion.aPumps[4].Linear.rActualPos;
GVL_HMI.stIOTerm26.rActualVelocity[1] 	:= GVL_Motion.aPumps[4].Linear.rActualVel;
GVL_HMI.stIOTerm26.rActualTorque[1] 	:= GVL_Motion.aPumps[4].Linear.rActualTorque;
GVL_HMI.stIOTerm26.bAxisHomed[1] 		:= GVL_Motion.aPumps[4].Linear.iHomed;
GVL_HMI.stIOTerm26.bAxisError[1] 		:= GVL_Motion.aPumps[4].Linear.iError;
GVL_HMI.stIOTerm26.nErrorCode[1] 		:= GVL_Motion.aPumps[4].Linear.nErrorCode;
GVL_HMI.stIOTerm26.bAxisOperational[2] 	:= GVL_Motion.aPumps[4].Rotary.iOperational;
GVL_HMI.stIOTerm26.rActualPosition[2] 	:= GVL_Motion.aPumps[4].Rotary.rActualPos;
GVL_HMI.stIOTerm26.rActualVelocity[2] 	:= GVL_Motion.aPumps[4].Rotary.rActualVel;
GVL_HMI.stIOTerm26.rActualTorque[2] 	:= GVL_Motion.aPumps[4].Rotary.rActualTorque;
GVL_HMI.stIOTerm26.bAxisHomed[2] 		:= GVL_Motion.aPumps[4].Rotary.iHomed;
GVL_HMI.stIOTerm26.bAxisError[2] 		:= GVL_Motion.aPumps[4].Rotary.iError;
GVL_HMI.stIOTerm26.nErrorCode[2] 		:= GVL_Motion.aPumps[4].Rotary.nErrorCode;

(* <EL7062 Terminal 27> -------------------------------------------------------------------------------------------------------------*)
GVL_HMI.stIOTerm27.bAxisOperational[1] 	:= GVL_Motion.aPumps[5].Linear.iOperational;
GVL_HMI.stIOTerm27.rActualPosition[1] 	:= GVL_Motion.aPumps[5].Linear.rActualPos;
GVL_HMI.stIOTerm27.rActualVelocity[1] 	:= GVL_Motion.aPumps[5].Linear.rActualVel;
GVL_HMI.stIOTerm27.rActualTorque[1] 	:= GVL_Motion.aPumps[5].Linear.rActualTorque;
GVL_HMI.stIOTerm27.bAxisHomed[1] 		:= GVL_Motion.aPumps[5].Linear.iHomed;
GVL_HMI.stIOTerm27.bAxisError[1] 		:= GVL_Motion.aPumps[5].Linear.iError;
GVL_HMI.stIOTerm27.nErrorCode[1] 		:= GVL_Motion.aPumps[5].Linear.nErrorCode;
GVL_HMI.stIOTerm27.bAxisOperational[2] 	:= GVL_Motion.aPumps[5].Rotary.iOperational;
GVL_HMI.stIOTerm27.rActualPosition[2] 	:= GVL_Motion.aPumps[5].Rotary.rActualPos;
GVL_HMI.stIOTerm27.rActualVelocity[2] 	:= GVL_Motion.aPumps[5].Rotary.rActualVel;
GVL_HMI.stIOTerm27.rActualTorque[2] 	:= GVL_Motion.aPumps[5].Rotary.rActualTorque;
GVL_HMI.stIOTerm27.bAxisHomed[2] 		:= GVL_Motion.aPumps[5].Rotary.iHomed;
GVL_HMI.stIOTerm27.bAxisError[2] 		:= GVL_Motion.aPumps[5].Rotary.iError;
GVL_HMI.stIOTerm27.nErrorCode[2] 		:= GVL_Motion.aPumps[5].Rotary.nErrorCode;

(* <EL7062 Terminal 28> -------------------------------------------------------------------------------------------------------------*)
GVL_HMI.stIOTerm28.bAxisOperational[1] 	:= GVL_Motion.aPumps[6].Linear.iOperational;
GVL_HMI.stIOTerm28.rActualPosition[1] 	:= GVL_Motion.aPumps[6].Linear.rActualPos;
GVL_HMI.stIOTerm28.rActualVelocity[1] 	:= GVL_Motion.aPumps[6].Linear.rActualVel;
GVL_HMI.stIOTerm28.rActualTorque[1] 	:= GVL_Motion.aPumps[6].Linear.rActualTorque;
GVL_HMI.stIOTerm28.bAxisHomed[1] 		:= GVL_Motion.aPumps[6].Linear.iHomed;
GVL_HMI.stIOTerm28.bAxisError[1] 		:= GVL_Motion.aPumps[6].Linear.iError;
GVL_HMI.stIOTerm28.nErrorCode[1] 		:= GVL_Motion.aPumps[6].Linear.nErrorCode;
GVL_HMI.stIOTerm28.bAxisOperational[2] 	:= GVL_Motion.aPumps[6].Rotary.iOperational;
GVL_HMI.stIOTerm28.rActualPosition[2] 	:= GVL_Motion.aPumps[6].Rotary.rActualPos;
GVL_HMI.stIOTerm28.rActualVelocity[2] 	:= GVL_Motion.aPumps[6].Rotary.rActualVel;
GVL_HMI.stIOTerm28.rActualTorque[2] 	:= GVL_Motion.aPumps[6].Rotary.rActualTorque;
GVL_HMI.stIOTerm28.bAxisHomed[2] 		:= GVL_Motion.aPumps[6].Rotary.iHomed;
GVL_HMI.stIOTerm28.bAxisError[2] 		:= GVL_Motion.aPumps[6].Rotary.iError;
GVL_HMI.stIOTerm28.nErrorCode[2] 		:= GVL_Motion.aPumps[6].Rotary.nErrorCode;

(* <EL7062 Terminal 29> -------------------------------------------------------------------------------------------------------------*)
GVL_HMI.stIOTerm29.bAxisOperational[1] 	:= GVL_Motion.aPumps[7].Linear.iOperational;
GVL_HMI.stIOTerm29.rActualPosition[1] 	:= GVL_Motion.aPumps[7].Linear.rActualPos;
GVL_HMI.stIOTerm29.rActualVelocity[1] 	:= GVL_Motion.aPumps[7].Linear.rActualVel;
GVL_HMI.stIOTerm29.rActualTorque[1] 	:= GVL_Motion.aPumps[7].Linear.rActualTorque;
GVL_HMI.stIOTerm29.bAxisHomed[1] 		:= GVL_Motion.aPumps[7].Linear.iHomed;
GVL_HMI.stIOTerm29.bAxisError[1] 		:= GVL_Motion.aPumps[7].Linear.iError;
GVL_HMI.stIOTerm29.nErrorCode[1] 		:= GVL_Motion.aPumps[7].Linear.nErrorCode;
GVL_HMI.stIOTerm29.bAxisOperational[2] 	:= GVL_Motion.aPumps[7].Rotary.iOperational;
GVL_HMI.stIOTerm29.rActualPosition[2] 	:= GVL_Motion.aPumps[7].Rotary.rActualPos;
GVL_HMI.stIOTerm29.rActualVelocity[2] 	:= GVL_Motion.aPumps[7].Rotary.rActualVel;
GVL_HMI.stIOTerm29.rActualTorque[2] 	:= GVL_Motion.aPumps[7].Rotary.rActualTorque;
GVL_HMI.stIOTerm29.bAxisHomed[2] 		:= GVL_Motion.aPumps[7].Rotary.iHomed;
GVL_HMI.stIOTerm29.bAxisError[2] 		:= GVL_Motion.aPumps[7].Rotary.iError;
GVL_HMI.stIOTerm29.nErrorCode[2] 		:= GVL_Motion.aPumps[7].Rotary.nErrorCode;

(* <EL7062 Terminal 30> -------------------------------------------------------------------------------------------------------------*)
GVL_HMI.stIOTerm30.bAxisOperational[1] 	:= GVL_Motion.aPumps[8].Linear.iOperational;
GVL_HMI.stIOTerm30.rActualPosition[1] 	:= GVL_Motion.aPumps[8].Linear.rActualPos;
GVL_HMI.stIOTerm30.rActualVelocity[1] 	:= GVL_Motion.aPumps[8].Linear.rActualVel;
GVL_HMI.stIOTerm30.rActualTorque[1] 	:= GVL_Motion.aPumps[8].Linear.rActualTorque;
GVL_HMI.stIOTerm30.bAxisHomed[1] 		:= GVL_Motion.aPumps[8].Linear.iHomed;
GVL_HMI.stIOTerm30.bAxisError[1] 		:= GVL_Motion.aPumps[8].Linear.iError;
GVL_HMI.stIOTerm30.nErrorCode[1] 		:= GVL_Motion.aPumps[8].Linear.nErrorCode;
GVL_HMI.stIOTerm30.bAxisOperational[2] 	:= GVL_Motion.aPumps[8].Rotary.iOperational;
GVL_HMI.stIOTerm30.rActualPosition[2] 	:= GVL_Motion.aPumps[8].Rotary.rActualPos;
GVL_HMI.stIOTerm30.rActualVelocity[2] 	:= GVL_Motion.aPumps[8].Rotary.rActualVel;
GVL_HMI.stIOTerm30.rActualTorque[2] 	:= GVL_Motion.aPumps[8].Rotary.rActualTorque;
GVL_HMI.stIOTerm30.bAxisHomed[2] 		:= GVL_Motion.aPumps[8].Rotary.iHomed;
GVL_HMI.stIOTerm30.bAxisError[2] 		:= GVL_Motion.aPumps[8].Rotary.iError;
GVL_HMI.stIOTerm30.nErrorCode[2] 		:= GVL_Motion.aPumps[8].Rotary.nErrorCode;

(* <EL7062 Terminal 31> -------------------------------------------------------------------------------------------------------------*)
GVL_HMI.stIOTerm31.bAxisOperational[1] 	:= GVL_Motion.aPumps[9].Linear.iOperational;
GVL_HMI.stIOTerm31.rActualPosition[1] 	:= GVL_Motion.aPumps[9].Linear.rActualPos;
GVL_HMI.stIOTerm31.rActualVelocity[1] 	:= GVL_Motion.aPumps[9].Linear.rActualVel;
GVL_HMI.stIOTerm31.rActualTorque[1] 	:= GVL_Motion.aPumps[9].Linear.rActualTorque;
GVL_HMI.stIOTerm31.bAxisHomed[1] 		:= GVL_Motion.aPumps[9].Linear.iHomed;
GVL_HMI.stIOTerm31.bAxisError[1] 		:= GVL_Motion.aPumps[9].Linear.iError;
GVL_HMI.stIOTerm31.nErrorCode[1] 		:= GVL_Motion.aPumps[9].Linear.nErrorCode;
GVL_HMI.stIOTerm31.bAxisOperational[2] 	:= GVL_Motion.aPumps[9].Rotary.iOperational;
GVL_HMI.stIOTerm31.rActualPosition[2] 	:= GVL_Motion.aPumps[9].Rotary.rActualPos;
GVL_HMI.stIOTerm31.rActualVelocity[2] 	:= GVL_Motion.aPumps[9].Rotary.rActualVel;
GVL_HMI.stIOTerm31.rActualTorque[2] 	:= GVL_Motion.aPumps[9].Rotary.rActualTorque;
GVL_HMI.stIOTerm31.bAxisHomed[2] 		:= GVL_Motion.aPumps[9].Rotary.iHomed;
GVL_HMI.stIOTerm31.bAxisError[2] 		:= GVL_Motion.aPumps[9].Rotary.iError;
GVL_HMI.stIOTerm31.nErrorCode[2] 		:= GVL_Motion.aPumps[9].Rotary.nErrorCode;

(* <EL7062 Terminal 32> -------------------------------------------------------------------------------------------------------------*)
GVL_HMI.stIOTerm32.bAxisOperational[1] 	:= GVL_Motion.aPumps[10].Linear.iOperational;
GVL_HMI.stIOTerm32.rActualPosition[1] 	:= GVL_Motion.aPumps[10].Linear.rActualPos;
GVL_HMI.stIOTerm32.rActualVelocity[1] 	:= GVL_Motion.aPumps[10].Linear.rActualVel;
GVL_HMI.stIOTerm32.rActualTorque[1] 	:= GVL_Motion.aPumps[10].Linear.rActualTorque;
GVL_HMI.stIOTerm32.bAxisHomed[1] 		:= GVL_Motion.aPumps[10].Linear.iHomed;
GVL_HMI.stIOTerm32.bAxisError[1] 		:= GVL_Motion.aPumps[10].Linear.iError;
GVL_HMI.stIOTerm32.nErrorCode[1] 		:= GVL_Motion.aPumps[10].Linear.nErrorCode;
GVL_HMI.stIOTerm32.bAxisOperational[2] 	:= GVL_Motion.aPumps[10].Rotary.iOperational;
GVL_HMI.stIOTerm32.rActualPosition[2] 	:= GVL_Motion.aPumps[10].Rotary.rActualPos;
GVL_HMI.stIOTerm32.rActualVelocity[2] 	:= GVL_Motion.aPumps[10].Rotary.rActualVel;
GVL_HMI.stIOTerm32.rActualTorque[2] 	:= GVL_Motion.aPumps[10].Rotary.rActualTorque;
GVL_HMI.stIOTerm32.bAxisHomed[2] 		:= GVL_Motion.aPumps[10].Rotary.iHomed;
GVL_HMI.stIOTerm32.bAxisError[2] 		:= GVL_Motion.aPumps[10].Rotary.iError;
GVL_HMI.stIOTerm32.nErrorCode[2] 		:= GVL_Motion.aPumps[10].Rotary.nErrorCode;

(* <EL7062 Terminal 34> -------------------------------------------------------------------------------------------------------------*)
GVL_HMI.stIOTerm34.bAxisOperational 	:= GVL_Motion.M1Motor.iOperational;
GVL_HMI.stIOTerm34.bAxisHomed 			:= GVL_Motion.M1Motor.iHomed;
GVL_HMI.stIOTerm34.bNotMoving			:= GVL_Motion.M1Motor.iNotMoving;
GVL_HMI.stIOTerm34.bAxisError 			:= GVL_Motion.M1Motor.iError;
GVL_HMI.stIOTerm34.bDriveError 			:= GVL_Motion.M1Motor.iError;
GVL_HMI.stIOTerm34.nErrorCode 			:= GVL_Motion.M1Motor.nErrorCode;
GVL_HMI.stIOTerm34.rActualPosition 		:= LINT_TO_LREAL(TRUNC(GVL_Motion.M1Motor.rActualPos * 1000)) /1000;
GVL_HMI.stIOTerm34.rActualVelocity 		:= LINT_TO_LREAL(TRUNC(GVL_Motion.M1Motor.rActualVel * 1000)) /1000;

(* <Box 1 ifm AL1333> --------------------------------------------------------------------------------------------------------------*)
GVL_HMI.aIOBox1[1] := GVL_HMI.HMIAnimation.aSolventLevel[1];
GVL_HMI.aIOBox1[2] := GVL_HMI.HMIAnimation.aSolventLevel[2];
GVL_HMI.aIOBox1[3] := GVL_HMI.HMIAnimation.aSolventLevel[3];
GVL_HMI.aIOBox1[4] := GVL_HMI.HMIAnimation.aSolventLevel[4];
GVL_HMI.aIOBox1[5] := GVL_HMI.HMIAnimation.rWasteLevel;

(* <Box 2 AMI8000 - Valve 1> -------------------------------------------------------------------------------------------------------------*)
GVL_HMI.aIOAMI8000[1].bAxisOperational 	:= GVL_Motion.aValves[1].iOperational;
GVL_HMI.aIOAMI8000[1].bAxisHomed 		:= GVL_Motion.aValves[1].iHomed;
GVL_HMI.aIOAMI8000[1].bNotMoving 		:= GVL_Motion.aValves[1].iNotMoving;
GVL_HMI.aIOAMI8000[1].bAxisError 		:= GVL_Motion.aValves[1].iError;
GVL_HMI.aIOAMI8000[1].nErrorCode 		:= GVL_Motion.aValves[1].nErrorCode;
GVL_HMI.aIOAMI8000[1].rActualPosition 	:= LINT_TO_LREAL(TRUNC(GVL_Motion.aValves[1].rActualPos* 1000)) /1000;
GVL_HMI.aIOAMI8000[1].rActualVelocity 	:= LINT_TO_LREAL(TRUNC(GVL_Motion.aValves[1].rActualVel* 1000)) /1000;

(* <Box 3 AMI8000 - Valve 2> -------------------------------------------------------------------------------------------------------------*)
GVL_HMI.aIOAMI8000[2].bAxisOperational 	:= GVL_Motion.aValves[2].iOperational;
GVL_HMI.aIOAMI8000[2].bAxisHomed 		:= GVL_Motion.aValves[2].iHomed;
GVL_HMI.aIOAMI8000[2].bNotMoving 		:= GVL_Motion.aValves[2].iNotMoving;
GVL_HMI.aIOAMI8000[2].bAxisError 		:= GVL_Motion.aValves[2].iError;
GVL_HMI.aIOAMI8000[2].nErrorCode 		:= GVL_Motion.aValves[2].nErrorCode;
GVL_HMI.aIOAMI8000[2].rActualPosition 	:= LINT_TO_LREAL(TRUNC(GVL_Motion.aValves[2].rActualPos* 1000)) /1000;
GVL_HMI.aIOAMI8000[2].rActualVelocity 	:= LINT_TO_LREAL(TRUNC(GVL_Motion.aValves[2].rActualVel* 1000)) /1000;

(* <Box 4 AMI8000 - Valve 3> -------------------------------------------------------------------------------------------------------------*)
GVL_HMI.aIOAMI8000[3].bAxisOperational 	:= GVL_Motion.aValves[3].iOperational;
GVL_HMI.aIOAMI8000[3].bAxisHomed 		:= GVL_Motion.aValves[3].iHomed;
GVL_HMI.aIOAMI8000[3].bNotMoving 		:= GVL_Motion.aValves[3].iNotMoving;
GVL_HMI.aIOAMI8000[3].bAxisError 		:= GVL_Motion.aValves[3].iError;
GVL_HMI.aIOAMI8000[3].nErrorCode 		:= GVL_Motion.aValves[3].nErrorCode;
GVL_HMI.aIOAMI8000[3].rActualPosition 	:= LINT_TO_LREAL(TRUNC(GVL_Motion.aValves[3].rActualPos* 1000)) /1000;
GVL_HMI.aIOAMI8000[3].rActualVelocity 	:= LINT_TO_LREAL(TRUNC(GVL_Motion.aValves[3].rActualVel* 1000)) /1000;

(* <Box 5 AMI8000 - Valve 4> -------------------------------------------------------------------------------------------------------------*)
GVL_HMI.aIOAMI8000[4].bAxisOperational 	:= GVL_Motion.aValves[4].iOperational;
GVL_HMI.aIOAMI8000[4].bAxisHomed 		:= GVL_Motion.aValves[4].iHomed;
GVL_HMI.aIOAMI8000[4].bNotMoving 		:= GVL_Motion.aValves[4].iNotMoving;
GVL_HMI.aIOAMI8000[4].bAxisError 		:= GVL_Motion.aValves[4].iError;
GVL_HMI.aIOAMI8000[4].nErrorCode 		:= GVL_Motion.aValves[4].nErrorCode;
GVL_HMI.aIOAMI8000[4].rActualPosition 	:= LINT_TO_LREAL(TRUNC(GVL_Motion.aValves[4].rActualPos* 1000)) /1000;
GVL_HMI.aIOAMI8000[4].rActualVelocity 	:= LINT_TO_LREAL(TRUNC(GVL_Motion.aValves[4].rActualVel* 1000)) /1000;

(* <Box 6 AMI8000 - Valve 5> -------------------------------------------------------------------------------------------------------------*)
GVL_HMI.aIOAMI8000[5].bAxisOperational 	:= GVL_Motion.aValves[5].iOperational;
GVL_HMI.aIOAMI8000[5].bAxisHomed 		:= GVL_Motion.aValves[5].iHomed;
GVL_HMI.aIOAMI8000[5].bNotMoving 		:= GVL_Motion.aValves[5].iNotMoving;
GVL_HMI.aIOAMI8000[5].bAxisError 		:= GVL_Motion.aValves[5].iError;
GVL_HMI.aIOAMI8000[5].nErrorCode 		:= GVL_Motion.aValves[5].nErrorCode;
GVL_HMI.aIOAMI8000[5].rActualPosition 	:= LINT_TO_LREAL(TRUNC(GVL_Motion.aValves[5].rActualPos* 1000)) /1000;
GVL_HMI.aIOAMI8000[5].rActualVelocity 	:= LINT_TO_LREAL(TRUNC(GVL_Motion.aValves[5].rActualVel* 1000)) /1000;

(* <Motors nState> -----------------------------------------------------------------------------------------------------------------*)
GVL_IO.nAX8108T34State := GVL_Motion.M1Motor.nState; //M1
GVL_IO.nEL7211T15State := GVL_Motion.M2Motor.nState; //M2
GVL_IO.nEL7211T16State := GVL_Motion.M3Motor.nState; //M3
GVL_IO.nAMI8000Box8State := GVL_Motion.aValves[1].nState; //Valve 1
GVL_IO.nAMI8000Box9State := GVL_Motion.aValves[2].nState; //Valve 2
GVL_IO.nAMI8000Box10State := GVL_Motion.aValves[3].nState; //Valve 3
GVL_IO.nAMI8000Box11State := GVL_Motion.aValves[4].nState; //Valve 4
GVL_IO.nAMI8000Box12State := GVL_Motion.aValves[5].nState; //Valve 5
GVL_IO.nEL7062T23State := GVL_Motion.aPumps[1].Linear.nState; //Pump1 Terminal
GVL_IO.nEL7062T24State := GVL_Motion.aPumps[2].Linear.nState; //Pump2 Terminal
GVL_IO.nEL7062T25State := GVL_Motion.aPumps[3].Linear.nState; //Pump3 Terminal
GVL_IO.nEL7062T26State := GVL_Motion.aPumps[4].Linear.nState; //Pump4 Terminal
GVL_IO.nEL7062T27State := GVL_Motion.aPumps[5].Linear.nState; //Pump5 Terminal
GVL_IO.nEL7062T28State := GVL_Motion.aPumps[6].Linear.nState; //Pump6 Terminal
GVL_IO.nEL7062T29State := GVL_Motion.aPumps[7].Linear.nState; //Pump7 Terminal
GVL_IO.nEL7062T30State := GVL_Motion.aPumps[8].Linear.nState; //Pump8 Terminal
GVL_IO.nEL7062T31State := GVL_Motion.aPumps[9].Linear.nState; //Pump9 Terminal
GVL_IO.nEL7062T32State := GVL_Motion.aPumps[10].Linear.nState; //Pump10 Terminal
END_ACTION

ACTION ACT_JarsAnimation:
(* Jar Animation *)

//when pumping into jars? Pump positive movement  

FOR i := 1 TO cJarsCount DO

    // ----------------- 1) Leitura posição (em VOLTAS) ------------------------
    curTurns := GVL_Motion.aPumps[i].Rotary.Axis.NcToPlc.ActPos / aUnitsPerTurn[i];

    // 2) Primeira amostra: inicializa e publica
    IF NOT aPrevInit[i] THEN
        aPrevTurns[i]     := curTurns;
        aPrevInit[i]      := TRUE;
        aDispMl[i]        := aJarMl[i];      // alinhar disp ao interno
        GVL_HMI.HmiAnimation.rJarFillAnimation[i] :=
            LIMIT(0.0, (aDispMl[i] / cJarCapacity_ml) * 100.0, 100.0);
        CONTINUE;
    END_IF

    // ----------------- 3) Delta e direção ------------------------------------
    deltaTurns := curTurns - aPrevTurns[i];
    dMl := deltaTurns * GVL_Motion.aPumps[i].Rotary.rPumpFactorFillJars;

    dir := 0;
    IF GVL_Motion.aPumps[i].Rotary.bPositiveDirection THEN
        dir := 1;
    ELSIF GVL_Motion.aPumps[i].Rotary.bNegativeDirection THEN
        dir := -1;
    ELSE
        IF dMl >  0.0 THEN dir := 1; END_IF
        IF dMl <  0.0 THEN dir := -1; END_IF
    END_IF

    // Sem movimento relevante?
    IF (ABS(deltaTurns) <= cEpsTurns) OR (dir = 0) THEN
        // publica (considerando se estava/está em recirculação)
        valIdx := ((i + 1) / 2); // 1&2->1, 3&4->2, ..., 9&10->5
        bRecircActive := (valIdx >= 1) AND (valIdx <= 5) AND
                         (GVL_Motion.aValves[valIdx].rActualPos >= cRecircLowDeg) AND
                         (GVL_Motion.aValves[valIdx].rActualPos <= cRecircHighDeg);

        IF bRecircActive THEN
            // sem movimento, mantém exibição atual (aDispMl)
        ELSE
            // fora da recirculação, exibe o interno
            aDispMl[i] := aJarMl[i];
        END_IF

        GVL_HMI.HmiAnimation.rJarFillAnimation[i] :=
            LIMIT(0.0, (aDispMl[i] / cJarCapacity_ml) * 100.0, 100.0);
        aPrevTurns[i] := curTurns;
        aRecircWasActive[i] := bRecircActive;
        CONTINUE;
    END_IF

    // ----------------- 4) Checar recirculação --------------------------------
    valIdx := ((i + 1) / 2);
    bRecircActive := (valIdx >= 1) AND (valIdx <= 5) AND
                     (GVL_Motion.aValves[valIdx].rActualPos >= cRecircLowDeg) AND
                     (GVL_Motion.aValves[valIdx].rActualPos <= cRecircHighDeg);

    IF bRecircActive THEN
        // Entrando agora? salva patamar base e sincroniza display
        IF NOT aRecircWasActive[i] THEN
            aRecircBaseMl[i] := aJarMl[i];     // patamar que “voltará” quando positivo
            aDispMl[i]       := aJarMl[i];     // start visual no nível atual
        END_IF

        // Anda a exibição “na razão da bomba”, sem alterar aJarMl
        IF dir < 0 THEN
            // cair até 20 mL gradualmente
            aDispMl[i] := MAX(cRecircDisplayMin_ml, aDispMl[i] - ABS(dMl));
        ELSIF dir > 0 THEN
            // subir de volta ao patamar base
            aDispMl[i] := MIN(aRecircBaseMl[i], aDispMl[i] + ABS(dMl));
        END_IF

        // Publicar exibição
        GVL_HMI.HmiAnimation.rJarFillAnimation[i] :=
            LIMIT(0.0, (aDispMl[i] / cJarCapacity_ml) * 100.0, 100.0);

        // Atualizações de referência e flags
        aPrevTurns[i]      := curTurns;
        aRecircWasActive[i]:= TRUE;

        // Pula integração/DeadVol: jar interno não muda em recirculação
        CONTINUE;
    END_IF

    // Saiu de recirculação agora? ressincroniza exibição com interno
    IF aRecircWasActive[i] AND (NOT bRecircActive) THEN
        aDispMl[i] := aJarMl[i];
    END_IF
    aRecircWasActive[i] := FALSE;

    // ----------------- 5) Lógica normal (fora da recirculação) ---------------
    // Mudou direção? novo segmento
    IF aSegDir[i] <> dir THEN
        aSegDir[i]       := dir;
        aSegAbsMl[i]     := 0.0;
        aSegAbsMlPrev[i] := 0.0;
    END_IF

    // Acumula módulo de mL neste segmento
    aSegAbsMlPrev[i] := aSegAbsMl[i];
    aSegAbsMl[i]     := aSegAbsMl[i] + ABS(dMl);

    // Aplica DeadVol por segmento:
    //  + Encher: só após exceder DeadVol o jar sobe
    //  - Esvaziar: só até (seg - DeadVol) o jar desce (últimos DeadVol não mexem)
    effDeltaMl := 0.0;

    IF dir = 1 THEN
        segNowEff  := MAX(0.0, aSegAbsMl[i]     - aDeadVolCfg_ml[i]);
        segPrevEff := MAX(0.0, aSegAbsMlPrev[i] - aDeadVolCfg_ml[i]);
        effDeltaMl := segNowEff - segPrevEff;        // aumenta jar
        aJarMl[i]  := aJarMl[i] + effDeltaMl;

    ELSIF dir = -1 THEN
        segNowEff  := MAX(0.0, aSegAbsMl[i]     - aDeadVolCfg_ml[i]);
        segPrevEff := MAX(0.0, aSegAbsMlPrev[i] - aDeadVolCfg_ml[i]);
        effDeltaMl := segNowEff - segPrevEff;        // diminui jar
        aJarMl[i]  := aJarMl[i] - effDeltaMl;
    END_IF

    // Limites físicos
    IF aJarMl[i] < 0.0 THEN aJarMl[i] := 0.0; END_IF
    IF aJarMl[i] > cJarCapacity_ml THEN aJarMl[i] := cJarCapacity_ml; END_IF

    // Publica (fora da recirculação, exibe o interno)
    aDispMl[i] := aJarMl[i];
    GVL_HMI.HmiAnimation.rJarFillAnimation[i] :=
        LIMIT(0.0, (aDispMl[i] / cJarCapacity_ml) * 100.0, 100.0);

    // Referência
    aPrevTurns[i] := curTurns;

END_FOR;
END_ACTION

ACTION ACT_M1Animation:
//M1 Motor vertical Axis Animation
IF GVL_Motion.bInitialHomingDone THEN
	// Read the end of scale value
	cM1MaxPosition := GVL_Settings.stMachineParam.aM1Position[2];	

	// Read motor Position
	rM1MotorPosition := GVL_Motion.M1Motor.rActualPos;
	
	//Check if cM1MaxPosition has a number different from 0
	IF cM1MaxPosition < 0 THEN
		// Scaling the motor position (0 = 0%, -320 = 100%)
		rM1MotorPositionPerc := ((rM1MotorPosition - cM1MinPosition) / (cM1MaxPosition - cM1MinPosition)) * 100.0; //Error 06/10/25
	ELSE
		rM1MotorPositionPerc := 0;
	END_IF
	
	// Limits value in the range 0 and 100%
	IF rM1MotorPositionPerc < 0 THEN
		rM1MotorPositionPerc := 0;
	ELSIF rM1MotorPositionPerc > 100 THEN
		rM1MotorPositionPerc := 100;
	END_IF
	
	GVL_HMI.HMIAnimation.rM1VerticalAnimation := 0 + (TO_REAL(rM1MotorPositionPerc)*1.55); //Adding y pixel home and sending the scaled value throug GVL_HMI
ELSE
	GVL_HMI.HMIAnimation.rM1VerticalAnimation := 0; //Default Value
END_IF
END_ACTION

ACTION ACT_M2Animation:
//M2 HMI object moves from pixel 455 (0 Position) up to 555 (Max position = -170mm)
//M2 Motor vertical Axis Animation
IF GVL_Motion.bInitialHomingDone THEN
	// Read the end of scale value
	cM2MaxPosition := GVL_Settings.stMachineParam.aM2Position[4]; //Calibration Position witch is the most away position the motor will reach	

	// Read motor Position
	rM2MotorPosition := GVL_Motion.M2Motor.rActualPos;
	
	//Check if cM2MaxPosition has a number different from 0
	IF cM2MaxPosition < 0 THEN
		// Scaling the motor position (0 = 0%, -320 = 100%)
		rM2MotorPositionPerc := ((rM2MotorPosition - cM2MinPosition) / (cM2MaxPosition - cM2MinPosition)) * 100.0; //Error 06/10/25
	ELSE
		rM2MotorPositionPerc := 0;
	END_IF
	
	// Limits value in the range 0 and 100%
	IF rM2MotorPositionPerc < 0 THEN
		rM2MotorPositionPerc := 0;
	ELSIF rM2MotorPositionPerc > 100 THEN
		rM2MotorPositionPerc := 100;
	END_IF
	
	GVL_HMI.HMIAnimation.rM2VerticalAnimation := 0 + (TO_REAL(rM2MotorPositionPerc)*0.9); //Adding y pixel home and sending the scaled value throug GVL_HMI
ELSE
	GVL_HMI.HMIAnimation.rM2VerticalAnimation := 0; //Default Value
END_IF
END_ACTION

END_PROGRAM

// ---- POUs/3. HMI/PRG_SaveSolvents.TcPOU
PROGRAM PRG_SaveSolvents
VAR
	rtSaveSolvents : R_TRIG;

	eState : (
		Idle,
		ValidateData,
		PrepareInsert,
		StartInsert,
		WaitInsertDone,
		Done,
		Error
	);

	i : INT;
	bValidationOk : BOOL;
END_VAR

rtSaveSolvents(CLK := GVL_HMI.bSaveSolventsBt);

CASE eState OF

	Idle:
		GVL_HMI.bSaveSolventsDone  := FALSE;
		GVL_HMI.bSaveSolventsError := FALSE;

		IF rtSaveSolvents.Q THEN
			eState := ValidateData;
		END_IF


	ValidateData:
		bValidationOk := TRUE;

		FOR i := 1 TO 4 DO

			IF GVL_HMI.stHMISolventsInfo[i].sSolventName = '' THEN
				bValidationOk := FALSE;
			END_IF

			IF GVL_HMI.stHMISolventsInfo[i].rDensity <= 0.0 THEN
				bValidationOk := FALSE;
			END_IF

		END_FOR

		IF bValidationOk THEN
			eState := PrepareInsert;
		ELSE
			eState := Error;
		END_IF


	PrepareInsert:
		GVL_DB.stSolvents.solventName1 := GVL_HMI.stHMISolventsInfo[1].sSolventName;
		GVL_DB.stSolvents.solventName2 := GVL_HMI.stHMISolventsInfo[2].sSolventName;
		GVL_DB.stSolvents.solventName3 := GVL_HMI.stHMISolventsInfo[3].sSolventName;
		GVL_DB.stSolvents.solventName4 := GVL_HMI.stHMISolventsInfo[4].sSolventName;

		GVL_DB.stSolvents.density1 := LREAL_TO_STRING(GVL_HMI.stHMISolventsInfo[1].rDensity);
		GVL_DB.stSolvents.density2 := LREAL_TO_STRING(GVL_HMI.stHMISolventsInfo[2].rDensity);
		GVL_DB.stSolvents.density3 := LREAL_TO_STRING(GVL_HMI.stHMISolventsInfo[3].rDensity);
		GVL_DB.stSolvents.density4 := LREAL_TO_STRING(GVL_HMI.stHMISolventsInfo[4].rDensity);

		GVL_DB.stSolvents.addedBy   := GVL_HMI.sUserNameEventTriggered;
		GVL_DB.stSolvents.addedDate := GVL_HMI.sDateAndTimeEventTriggered;

		eState := StartInsert;


	StartInsert:
		IF DB_Query.state = E_DB_QUERY_STATE.IDLE_STATE THEN
			DB_Query.state := E_DB_QUERY_STATE.INSERT_SOLVENT;
			eState := WaitInsertDone;
		END_IF


	WaitInsertDone:
		IF DB_Query.state = E_DB_QUERY_STATE.ERROR_STATE THEN
			eState := Error;

		ELSIF (DB_Query.state = E_DB_QUERY_STATE.IDLE_STATE) AND NOT DB_Query.bBusyDb THEN

			// Update the runtime settings only after successful DB insert
			GVL_Settings.stSolventsInfo := GVL_HMI.stHMISolventsInfo;

			GVL_HMI.bSaveSolventsDone := TRUE;
			GVL_HMI.bSaveSolventsBt   := FALSE;

			eState := Done;
		END_IF


	Done:
		eState := Idle;


	Error:
		GVL_HMI.bSaveSolventsError := TRUE;
		GVL_HMI.bSaveSolventsBt    := FALSE;
		eState := Idle;

END_CASE

END_PROGRAM

// ---- POUs/Utilities/PRG_TowerAlarmLamps.TcPOU
PROGRAM PRG_TowerAlarmLamps
VAR
	fbBlinkRedLight, fbBlinkAmbarLight, fbBlinkGreenLight	: FB_Blink; //Flashing lights FB
	
END_VAR

// Reset all tower lights and blinkers to a safe state before setting according to mode
GVL_IO.gDigOutputs.bTowerGreenLight := FALSE;
GVL_IO.gDigOutputs.bTowerAmberLight := FALSE;
GVL_IO.gDigOutputs.bTowerRedLight := FALSE;
//fbBlinkRedLight(bEnable := FALSE, tPeriod := T#500MS);
//fbBlinkAmbarLight(bEnable := FALSE, tPeriod := T#500MS);

CASE GVL_HMI.eMachineMode OF

    E_MachineMode.AUTO_CYCLE:
        // Green steady
        GVL_IO.gDigOutputs.bTowerGreenLight := TRUE;

    E_MachineMode.CALIBRATION:
        // Amber steady
        GVL_IO.gDigOutputs.bTowerAmberLight := TRUE;

    E_MachineMode.IMEDIATE_FAULT:
        // Red flashing
        fbBlinkRedLight(bEnable := TRUE, tPeriod := T#1S);
        GVL_IO.gDigOutputs.bTowerRedLight := fbBlinkRedLight.bBlink;

    E_MachineMode.MANUAL:
        // Amber steady
        GVL_IO.gDigOutputs.bTowerAmberLight := TRUE;

    E_MachineMode.STOPPED:
        // Red steady
        GVL_IO.gDigOutputs.bTowerRedLight := TRUE;
	
	E_MachineMode.SYSTEM_INITIALIZING:
		// Amber flashing
        fbBlinkAmbarLight(bEnable := TRUE, tPeriod := T#1S);
        GVL_IO.gDigOutputs.bTowerAmberLight := fbBlinkAmbarLight.bBlink;
	
	E_MachineMode.SYSTEM_READY:
		// Green flashing
        fbBlinkGreenLight(bEnable := TRUE, tPeriod := T#1S);
        GVL_IO.gDigOutputs.bTowerGreenLight := fbBlinkGreenLight.bBlink;

    ELSE
        // Unknown state - All lights off
        GVL_IO.gDigOutputs.bTowerGreenLight := FALSE;
        GVL_IO.gDigOutputs.bTowerAmberLight := FALSE;
        GVL_IO.gDigOutputs.bTowerRedLight := FALSE;
        fbBlinkRedLight(bEnable := FALSE, tPeriod := T#500MS);
        fbBlinkAmbarLight(bEnable := FALSE, tPeriod := T#500MS);
END_CASE

END_PROGRAM

// ---- POUs/Levels/PRG_LevelHandler.TcPOU
PROGRAM PRG_LevelHandler
VAR
	fbParser : ARRAY[1..5] OF FB_KQ1000_Parser;
    stLevels : ARRAY[1..5] OF ST_KQ1000_Data;
	
	rRinseLevel : ARRAY[1..4] OF REAL;
	rWasteLevel : REAL;

	//Variables Mapping from ifm AL1333	
	
	// Ch1 = Rinse 1 bottle
    byCh1_0 AT %IB0 : BYTE;
    byCh1_1 AT %IB1 : BYTE;
    byCh1_2 AT %IB2 : BYTE;
    byCh1_3 AT %IB3 : BYTE;
	
	// Ch2 = Rinse 2 bottle
    byCh2_0 AT %IB4 : BYTE;
    byCh2_1 AT %IB5 : BYTE;
    byCh2_2 AT %IB6 : BYTE;
    byCh2_3 AT %IB7 : BYTE;
	
	// Ch3 = Rinse 3 bottle
    byCh3_0 AT %IB8 : BYTE;
    byCh3_1 AT %IB9 : BYTE;
    byCh3_2 AT %IB10 : BYTE;
    byCh3_3 AT %IB11 : BYTE;
	
	// Ch4 = Rinse 4 bottle
    byCh4_0 AT %IB12 : BYTE;
    byCh4_1 AT %IB13 : BYTE;
    byCh4_2 AT %IB14 : BYTE;
    byCh4_3 AT %IB15 : BYTE;
	
	// Ch5 = Waste Container
    byCh5_0 AT %IB16 : BYTE;
    byCh5_1 AT %IB17 : BYTE;
    byCh5_2 AT %IB18 : BYTE;
    byCh5_3 AT %IB19 : BYTE;
	
	bRinseBottle1_OK   : BOOL := (stLevels[1].rLevelPercent >= 10.0); // Exemplo de condição
	iWasteDeviceStatus : USINT := stLevels[5].iDeviceStatusCode;

	
END_VAR

// Execute the parsers
fbParser[1](byInput0 := byCh1_0, byInput1 := byCh1_1, byInput2 := byCh1_2, byInput3 := byCh1_3);
stLevels[1] := fbParser[1].stData;
rRinseLevel[1] := stLevels[1].rLevelPercent;

fbParser[2](byInput0 := byCh2_0, byInput1 := byCh2_1, byInput2 := byCh2_2, byInput3 := byCh2_3);
stLevels[2] := fbParser[2].stData;
rRinseLevel[2] := stLevels[2].rLevelPercent;

fbParser[3](byInput0 := byCh3_0, byInput1 := byCh3_1, byInput2 := byCh3_2, byInput3 := byCh3_3);
stLevels[3] := fbParser[3].stData;
rRinseLevel[3] := stLevels[3].rLevelPercent;

fbParser[4](byInput0 := byCh4_0, byInput1 := byCh4_1, byInput2 := byCh4_2, byInput3 := byCh4_3);
stLevels[4] := fbParser[4].stData;
rRinseLevel[4] := stLevels[4].rLevelPercent;

fbParser[5](byInput0 := byCh5_0, byInput1 := byCh5_1, byInput2 := byCh5_2, byInput3 := byCh5_3);
stLevels[5] := fbParser[5].stData;
rWasteLevel := stLevels[5].rLevelPercent;

//Update HMI bottles animation
GVL_HMI.HMIAnimation.aSolventLevel[1]	:= TO_INT(rRinseLevel[1]);
GVL_HMI.HMIAnimation.aSolventLevel[2]	:= TO_INT(rRinseLevel[2]);
GVL_HMI.HMIAnimation.aSolventLevel[3]	:= TO_INT(rRinseLevel[3]);
GVL_HMI.HMIAnimation.aSolventLevel[4]	:= TO_INT(rRinseLevel[4]);
GVL_HMI.HMIAnimation.rWasteLevel		:= TO_INT(rWasteLevel);

(* Levels Process Warnings Logic *) //--------------------------------------------------------------------------------------------

// Flag to warning when solvent reservoirs are bellow 50% level
IF GVL_HMI.HMIAnimation.aSolventLevel[1] <= 50 THEN
	GVL_Alarms.aSolventNearLowLevel[1] := TRUE;
ELSE
	GVL_Alarms.aSolventNearLowLevel[1] := FALSE;
END_IF

IF GVL_HMI.HMIAnimation.aSolventLevel[2] <= 50 THEN
	GVL_Alarms.aSolventNearLowLevel[2] := TRUE;
ELSE
	GVL_Alarms.aSolventNearLowLevel[2] := FALSE;
END_IF

IF GVL_HMI.HMIAnimation.aSolventLevel[3] <= 50 THEN
	GVL_Alarms.aSolventNearLowLevel[3] := TRUE;
ELSE
	GVL_Alarms.aSolventNearLowLevel[3] := FALSE;
END_IF

IF GVL_HMI.HMIAnimation.aSolventLevel[4] <= 50 THEN
	GVL_Alarms.aSolventNearLowLevel[4] := TRUE;
ELSE
	GVL_Alarms.aSolventNearLowLevel[4] := FALSE;
END_IF

// Flag to warning when waste reservoirs are above 60% level
IF GVL_HMI.HMIAnimation.rWasteLevel >= 60 THEN
	GVL_Alarms.bWasteNearHighLevel := TRUE;
ELSE
	GVL_Alarms.bWasteNearHighLevel := FALSE;
END_IF

END_PROGRAM

// ---- POUs/Levels/FB_KQ1000_Parser.TcPOU
FUNCTION_BLOCK FB_KQ1000_Parser
VAR_INPUT
	byInput0 : BYTE;
    byInput1 : BYTE;
    byInput2 : BYTE;
    byInput3 : BYTE;
END_VAR
VAR_OUTPUT
	stData : ST_KQ1000_Data;
END_VAR
VAR
	wLevel	: WORD;
    wStatus : WORD;
END_VAR

// Combine the bytes to form the full raw level word
wLevel := SHL(TO_WORD(byInput1), 8) OR TO_WORD(byInput0);

// Check for NoData condition (specific code from sensor)
IF wLevel = 32764 THEN
    stData.iRawLevel := wLevel;
    stData.rLevelPercent := -1.0;
ELSE
    // Store the visible base level (based on byte 1 only)
    stData.iRawLevel := TO_WORD(byInput1);

    // Linear scaling: 10 = 0%, 95 = 100%
    IF byInput1 < 10 THEN
        stData.rLevelPercent := 0.0;
    ELSIF byInput1 > 95 THEN
        stData.rLevelPercent := 100.0;
    ELSE
        stData.rLevelPercent := (TO_REAL(byInput1 - 5) * (100.0 / 85.0)); 
    END_IF
END_IF

// Combine bytes to get the full status word
wStatus := SHL(TO_WORD(byInput3), 8) OR TO_WORD(byInput2);
stData.wStatusRaw := wStatus;

// Decode output status bits
stData.bOut1 := (wStatus AND 16#0001) <> 0;
stData.bOut2 := (wStatus AND 16#0002) <> 0;
stData.bOut3 := (wStatus AND 16#0004) <> 0;

// Extract device status code from bits 4–7
stData.iDeviceStatusCode := TO_USINT(SHR(wStatus AND 16#00F0, 4));

END_FUNCTION_BLOCK

// ---- POUs/6. Reports/PRG_ReportsManager.TcPOU
PROGRAM PRG_ReportsManager
VAR
	rTrigPdfConsumed : R_TRIG;
END_VAR

rTrigPdfConsumed(CLK := GVL_Reports.bPdfConsumed);

IF rTrigPdfConsumed.Q THEN
    GVL_Reports.bLoadDone      	 := FALSE;
    GVL_Reports.bLoadBusy      	 := FALSE;
    GVL_Reports.bLoadError     	 := FALSE;
    GVL_Reports.bPdfDataReady  	 := FALSE;
    GVL_Reports.bPdfConsumed   	 := FALSE;
    GVL_Reports.sLoadStatus    	 := 'Idle';
	GVL_Reports.sQuickReportName := '';
END_IF

IF GVL_Reports.bClearSearchScreen THEN
    GVL_Reports.bClearSearchScreen := FALSE;
    Clear_ReportsListing();
END_IF

IF GVL_Reports.bBuildCurrentLinearReport THEN
    GVL_Reports.bBuildCurrentLinearReport := FALSE;
	GVL_Reports.eSelectedReportType := E_ReportType.LinearMotors;
    DB_Query.state := E_DB_QUERY_STATE.SELECT_LAST_LINEAR_REPORT;
END_IF

IF GVL_Reports.bBuildLastPostRunReport THEN
    GVL_Reports.bBuildLastPostRunReport := FALSE;
    GVL_Reports.eSelectedReportType := E_ReportType.PostRun;
    DB_Query.state := E_DB_QUERY_STATE.SELECT_LAST_POSTRUN_RUN;
END_IF

IF GVL_Reports.bBuildLastPumpCalibrationReport THEN
    GVL_Reports.bBuildLastPumpCalibrationReport := FALSE;
    GVL_Reports.eSelectedReportType := E_ReportType.PumpCalibration;
    GVL_Reports.sQuickReportName := '';
    DB_Query.state := E_DB_QUERY_STATE.SELECT_LAST_PUMP_CALIBRATION;
END_IF

IF GVL_Reports.bBuildSystemHistoryReport THEN
    GVL_Reports.bBuildSystemHistoryReport := FALSE;
    GVL_Reports.eSelectedReportType := E_ReportType.SystemSettings;
    GVL_Reports.sQuickReportName := 'SystemHistory';
    DB_Query.state := E_DB_QUERY_STATE.SELECT_SYSTEM_HISTORY_REPORT;
END_IF

IF GVL_Reports.bBuildLinearHistoryReport THEN
    GVL_Reports.bBuildLinearHistoryReport := FALSE;
    GVL_Reports.eSelectedReportType := E_ReportType.LinearMotors;
    GVL_Reports.sQuickReportName := 'LinearHistory';
    DB_Query.state := E_DB_QUERY_STATE.SELECT_LINEAR_HISTORY_REPORT;
END_IF


IF GVL_Reports.bBuildCompleteMethodReport THEN
    GVL_Reports.bBuildCompleteMethodReport := FALSE;
    GVL_Reports.eSelectedReportType := E_ReportType.Recipe;
    GVL_Reports.sQuickReportName := 'CompleteMethodHistory';
    DB_Query.state := E_DB_QUERY_STATE.SELECT_COMPLETE_METHOD_REPORT;
END_IF

IF GVL_Reports.bLoadSelectedReport THEN
    GVL_Reports.bLoadSelectedReport := FALSE;

    CASE GVL_Reports.eSelectedReportType OF
        E_ReportType.PumpCalibration:
            DB_Query.state := E_DB_QUERY_STATE.SELECT_CALIB_REPORT_BY_ID;

        E_ReportType.SystemSettings:
            DB_Query.state := E_DB_QUERY_STATE.SELECT_SYSTEM_SETTINGS_BY_ID;

        E_ReportType.Recipe:
            // Recipe reports load by methodID stored in sSelectedPrimaryID.
            // NOTE: Add SELECT_RECIPE_REPORT_BY_ID to E_DB_QUERY_STATE and
            // implement the state in DB_Query if detailed recipe PDF is needed.
			DB_Query.state := E_DB_QUERY_STATE.SELECT_RECIPE_HEADER_BY_ID;
            GVL_Reports.bPdfDataReady := TRUE;
            GVL_Reports.bPdfConsumed  := FALSE;

        E_ReportType.PostRun:
            // PostRun reports load by runNo stored in sSelectedPrimaryID.
            // NOTE: Add SELECT_RUN_REPORT_BY_ID to E_DB_QUERY_STATE and
            // implement the state in DB_Query if detailed run PDF is needed.
			DB_Query.state := E_DB_QUERY_STATE.SELECT_POSTRUN_RUN_BY_ID;
            GVL_Reports.bPdfDataReady := TRUE;
            GVL_Reports.bPdfConsumed  := FALSE;
		
		E_ReportType.LinearMotors:
  			DB_Query.state := E_DB_QUERY_STATE.SELECT_LINEAR_BY_ID;

    ELSE
        GVL_Reports.bLoadError  := TRUE;
        GVL_Reports.bLoadBusy   := FALSE;
        GVL_Reports.bLoadDone   := FALSE;
        GVL_Reports.sLoadStatus := 'Invalid report type selected';
    END_CASE
END_IF


IF GVL_Reports.bSearchRequest THEN
    GVL_Reports.bSearchRequest := FALSE;

    DB_Query.Clear_ReportSearchResult();

    CASE GVL_Reports.eSelectedReportType OF
        E_ReportType.PumpCalibration:
            DB_Query.state := E_DB_QUERY_STATE.SELECT_CALIB_REPORT_LIST;

        E_ReportType.SystemSettings:
            DB_Query.state := E_DB_QUERY_STATE.SELECT_SYSTEM_SETTINGS_REPORT_LIST;

        E_ReportType.Recipe:
            DB_Query.state := E_DB_QUERY_STATE.SELECT_METHOD_REPORT_SEARCH;

        E_ReportType.PostRun:
            DB_Query.state := E_DB_QUERY_STATE.SELECT_RUN_REPORT_LIST;
		
		E_ReportType.LinearMotors:
			
			DB_Query.state := E_DB_QUERY_STATE.SELECT_LINEAR_REPORT_SEARCH;

    ELSE
        GVL_Reports.bSearchBusy   := FALSE;
        GVL_Reports.bSearchDone   := FALSE;
        GVL_Reports.bSearchError  := TRUE;
        GVL_Reports.sSearchStatus := 'Could not prepare report search.';
    END_CASE
END_IF

METHOD Clear_ReportsListing : BOOL
VAR_INPUT
END_VAR
GVL_Reports.bClearSearchScreen := FALSE;

DB_Query.Clear_ReportSearchResult();

GVL_Reports.eSelectedReportType := E_ReportType.None;
GVL_Reports.sSelectedPrimaryID  := '';
GVL_Reports.sSelectedReportName := '';

GVL_Reports.uiReportSearchCount := 0;
GVL_Reports.bSearchRequest      := FALSE;
GVL_Reports.bSearchBusy         := FALSE;
GVL_Reports.bSearchDone         := FALSE;
GVL_Reports.bSearchError        := FALSE;
GVL_Reports.sSearchStatus       := 'Idle';

GVL_Reports.bLoadSelectedReport := FALSE;
GVL_Reports.bLoadBusy           := FALSE;
GVL_Reports.bLoadDone           := FALSE;
GVL_Reports.bLoadError          := FALSE;
GVL_Reports.bPdfDataReady       := FALSE;
GVL_Reports.bPdfConsumed        := FALSE;
GVL_Reports.sLoadStatus         := 'Idle';
END_METHOD

END_PROGRAM

// ---- POUs/4. RecipeHandle/PRG_RecipeManager.TcPOU
PROGRAM PRG_RecipeManager
VAR
	fbLoadRecipe  	: FB_LoadRecipe;
    fbListFiles  	: FB_ListRecipeFiles;
	fbDeleteRecipe 	: FB_DeleteRecipe;
	fbSaveRecipe 	: FB_SaveRecipe;

    sPrefix      : STRING(64) := 'C:\TwinCAT\Recipes\';
    sFileName    : STRING(255);
	
	bDatagridRowsNaming		 : BOOL := FALSE;
	bClearAvailableFiles	 : BOOL := FALSE;
	bClearAvailableFilesDone : BOOL := FALSE;
	
	
		
	i	: INT;
	
	
END_VAR

VAR_INPUT
	bDatagridToRecipeDone	: BOOL := FALSE;
END_VAR

//Naming the datagrid 1st column with the names in the HMI Recipe Screen just once
IF NOT bDatagridRowsNaming THEN
	ACT_DatagridsRowNaming();
END_IF

// <Load button> ############# Look up for the recipe files in the folder and fill up the GVL_Recipe.aAvailableFiles[]. ######################### 
IF GVL_HMI.bRefreshRecipeList THEN
	//GVL_HMI.bRecipeCorrectLoaded := FALSE;
	//GVL_HMI.bRecipeLoadFailed := FALSE;
	bClearAvailableFiles := TRUE;
	IF bClearAvailableFilesDone THEN
		fbListFiles(bExecute := TRUE);
	END_IF
ELSE
	bClearAvailableFiles := FALSE;
	bClearAvailableFilesDone := FALSE;
    fbListFiles(bExecute := FALSE);
END_IF

// Clear the Available files datagrid in the load file popup
IF bClearAvailableFiles THEN
	ACT_ClearAvailableFiles();
END_IF

// Reset load actions once its done
IF fbListFiles.bDone THEN
	GVL_HMI.bRefreshRecipeList := FALSE;
END_IF

 //Reset file name
sFileName := '';

// Run the loading recipe from selected row in the recipe load popup
sFileName := CONCAT(sPrefix, CONCAT(GVL_Recipe.sSelectedRecipeName, '.json')); // File naming assemble for the selected row in the recipe load popup
fbLoadRecipe( sFileName := sFileName, bExecute := GVL_HMI.bRecipeLoadFromFile AND  DB_Query.timerVD.Q );


IF fbLoadRecipe.bError THEN
	GVL_HMI.bRecipeLoadFailed := TRUE;
	//GVL_HMI.bRecipeLoadFromFile := FALSE;
END_IF

// After the recipe loading, reseting and setting the flags
IF NOT fbLoadRecipe.bBusy AND NOT fbLoadRecipe.bError AND GVL_HMI.bRecipeLoadFromFile AND DB_Query.timerVD.Q THEN
	GVL_HMI.bRecipeCorrectLoaded := TRUE;
	GVL_HMI.bRecipeLoadFromFile := FALSE;
	DB_Query.timerVD(in:= FALSE);
	ACT_ClearStActiveRecipe(); //Clears the Active Recipe
END_IF
// <\Load button> ############# END ##############

// <Save Button> ############# Fill stCurrentRecipe from HMI datagrids if save button is pressed ########################
IF GVL_HMI.bRecipeSaveButton THEN
	ACT_DatagridToRecipe();
	IF bDatagridToRecipeDone THEN
		fbSaveRecipe(bExecute := TRUE, sUser := GVL_HMI.stRecipeInfo.sCreatedBy);
		IF fbSaveRecipe.bDone AND NOT fbSaveRecipe.bError THEN
			GVL_HMI.stRecipeInfo.iRevision := GVL_Recipe.stCurrentRecipe.stInfo.iRevision; //Update the datagrid revision that does not come from the grid
			fbSaveRecipe(bExecute := FALSE);
			//GVL_HMI.bRecipeSaveDone := true; //Response Success flag to HMI // chenged 13/11/25
			GVL_HMI.bRecipeSaveButton := FALSE;	
			bDatagridToRecipeDone := FALSE;
			ACT_ClearStActiveRecipe(); //Clears the Active Recipe
			ELSE IF fbSaveRecipe.bError THEN
				GVL_HMI.bRecipeSaveError := TRUE; //Response Error flag to HMI
			END_IF
		END_IF
		
	END_IF
END_IF
// <\Save Button> ############# END ########################

// <Cancel Button> ############# Reload the datagrids with the recipe in stCurrentRecipe if the bt cancel is pressed during new recipe ########################
IF GVL_HMI.bReloadRecipeDatagrids THEN
	ACT_RecipeToDatagrid();
END_IF
// <\Cancel Button> ############# END ########################

// <Activate Button> ############# Transfer data from stCurrentRecipe for stActivatedRecipe witch will be used on the cycle  ########################
IF GVL_HMI.bRecipeActivateButton THEN
	GVL_Recipe.stActiveRecipe := GVL_Recipe.stCurrentRecipe; //Only fill stActiveRecipe if button Activate was pressed on hmi. 
	IF GVL_Recipe.stCurrentRecipe.stInfo.sMethodName <> '' THEN
		GVL_HMI.bRecipeActivateDone := TRUE;
		GVL_Recipe.bIsThereRecipeActivated := TRUE;
	ELSE
		GVL_HMI.bRecipeActivateError := TRUE;
	END_IF
	
END_IF
// <\Activate Button> ############# END ########################

// <Delete Button> ############# Moves the loaded Recipe file from the root folder for the _deleted folder ########################
IF GVL_HMI.bDeleteRecipeButton THEN
	ACT_PopulateDeleteRecipeInfo();
	GVL_HMI.bDeleteRecipeDone := FALSE;
	GVL_HMI.bDeleteRecipeError := FALSE;
END_IF

fbDeleteRecipe(bExecute := GVL_HMI.bDeleteRecipeConfirm, stFileInfo := GVL_HMI.stDeleteRecipeInfo);

IF fbDeleteRecipe.bDone THEN
	IF NOT fbDeleteRecipe.bError THEN 
		ACT_ClearStCurrentRecipe();
		ACT_ClearHMIDatagrids();
		ACT_ClearStActiveRecipe(); //Clears the Active Recipe
		GVL_HMI.bDeleteRecipeConfirm := FALSE;
		GVL_HMI.bDeleteRecipeDone := TRUE;
	ELSE 
		GVL_HMI.bDeleteRecipeError := TRUE;
	END_IF
END_IF

// <\Delete Button> ############# END ########################

ACTION ACT_ClearAvailableFiles:
//Clear the GVL_Recipe.aAvailableFiles, witch is the list files datagrid data source
IF NOT bClearAvailableFilesDone THEN
	FOR i := 1 TO 50 DO
		GVL_HMI.aAvailableFiles[i].sFileName := '';
		GVL_HMI.aAvailableFiles[i].sMethodName := '';
		GVL_HMI.aAvailableFiles[i].sCreatedBy := '';
		GVL_HMI.aAvailableFiles[i].iRevision := 0;
		GVL_HMI.aAvailableFiles[i].dtLastModified := DT#1970-01-01-00:00;
		GVL_HMI.aAvailableFiles[i].dCreationDate := D#1970-01-01;
	END_FOR
	
	IF i >= 50 THEN
		bClearAvailableFilesDone := TRUE;
	END_IF
END_IF
END_ACTION

ACTION ACT_ClearHMIDatagrids:
//Clear the arrays that are binding with the datagrids source on recipe HMI content
//Recipe Info fields
GVL_HMI.stRecipeInfo.dCreationDate := D#1970-01-01;
GVL_HMI.stRecipeInfo.iRevision := 0;
GVL_HMI.stRecipeInfo.sCreatedBy := '';
GVL_HMI.stRecipeInfo.sMethodName := '';

//Solvents and Times datagrid
FOR i := 1 TO 3 DO
	GVL_HMI.aSolventAndTimesRows[i].Rinse1 := 0;
	GVL_HMI.aSolventAndTimesRows[i].Rinse2 := 0;
	GVL_HMI.aSolventAndTimesRows[i].Wash1 := 0;
	GVL_HMI.aSolventAndTimesRows[i].Wash2 := 0;
END_FOR

//Volumes datagrid
FOR i := 1 TO 10 DO
	GVL_HMI.aVolumeRows[i].Rinse1 := 0;
	GVL_HMI.aVolumeRows[i].Rinse2 := 0;
	GVL_HMI.aVolumeRows[i].Wash1 := 0;
	GVL_HMI.aVolumeRows[i].Wash2 := 0;
END_FOR

//Other Parameters datagrid
FOR i := 1 TO 8 DO
	GVL_HMI.aOtherParamsRows[i].Value := 0;
END_FOR
END_ACTION

ACTION ACT_ClearStActiveRecipe:
//Clear Flags 
GVL_Recipe.bIsThereRecipeActivated := FALSE;
GVL_HMI.bRecipeActivateDone := FALSE;
GVL_HMI.bRecipeActivateError := FALSE;
//Clears the array stCurrentRecipe 
//Info
GVL_Recipe.stActiveRecipe.stInfo.dCreationDate := D#1970-01-01;
GVL_Recipe.stActiveRecipe.stInfo.iRevision := 0;
GVL_Recipe.stActiveRecipe.stInfo.sCreatedBy := '';
GVL_Recipe.stActiveRecipe.stInfo.sMethodName := '';


//Other Parameters
GVL_Recipe.stActiveRecipe.stOtherParams.iVialsToFill := 0;
GVL_Recipe.stActiveRecipe.stOtherParams.rVial1FillVol := 0;
GVL_Recipe.stActiveRecipe.stOtherParams.rVialPrimeVol := 0;
GVL_Recipe.stActiveRecipe.stOtherParams.rVials2_4FillVol := 0;
GVL_Recipe.stActiveRecipe.stOtherParams.tAgitate1Time := T#0S;
GVL_Recipe.stActiveRecipe.stOtherParams.tAgitate2Time := T#0S;
GVL_Recipe.stActiveRecipe.stOtherParams.tAirDryTime := T#0S;
GVL_Recipe.stActiveRecipe.stOtherParams.tSoakTime := T#0S;

FOR i := 1 TO 4 DO
	//Solvents and Times
	GVL_Recipe.stActiveRecipe.stSolventsTimes.aSolventN[i] := 0;
	GVL_Recipe.stActiveRecipe.stSolventsTimes.aTime[i] := T#0S;
	GVL_Recipe.stActiveRecipe.stSolventsTimes.aVelocity[i] := 0;
	
	//Volumes
	GVL_Recipe.stActiveRecipe.stVolumes.aF_Volume[i] := 0;
	GVL_Recipe.stActiveRecipe.stVolumes.aS0_Volume[i] := 0;
	GVL_Recipe.stActiveRecipe.stVolumes.aS1_Volume[i] := 0;
	GVL_Recipe.stActiveRecipe.stVolumes.aS2_Volume[i] := 0;
	GVL_Recipe.stActiveRecipe.stVolumes.aS3_Volume[i] := 0;
	GVL_Recipe.stActiveRecipe.stVolumes.aS4_Volume[i] := 0;
	GVL_Recipe.stActiveRecipe.stVolumes.aS5_Volume[i] := 0;
	GVL_Recipe.stActiveRecipe.stVolumes.aS6_Volume[i] := 0;
	GVL_Recipe.stActiveRecipe.stVolumes.aS7_Volume[i] := 0;
	GVL_Recipe.stActiveRecipe.stVolumes.aT_IC_Volume[i] := 0;
END_FOR
END_ACTION

ACTION ACT_ClearStCurrentRecipe:
//Clears the array stCurrentRecipe 
//Info
GVL_Recipe.stCurrentRecipe.stInfo.dCreationDate := D#1970-01-01;
GVL_Recipe.stCurrentRecipe.stInfo.iRevision := 0;
GVL_Recipe.stCurrentRecipe.stInfo.sCreatedBy := '';
GVL_Recipe.stCurrentRecipe.stInfo.sMethodName := '';

//Other Parameters
GVL_Recipe.stCurrentRecipe.stOtherParams.iVialsToFill := 0;
GVL_Recipe.stCurrentRecipe.stOtherParams.rVial1FillVol := 0;
GVL_Recipe.stCurrentRecipe.stOtherParams.rVialPrimeVol := 0;
GVL_Recipe.stCurrentRecipe.stOtherParams.rVials2_4FillVol := 0;
GVL_Recipe.stCurrentRecipe.stOtherParams.tAgitate1Time := T#0S;
GVL_Recipe.stCurrentRecipe.stOtherParams.tAgitate2Time := T#0S;
GVL_Recipe.stCurrentRecipe.stOtherParams.tAirDryTime := T#0S;
GVL_Recipe.stCurrentRecipe.stOtherParams.tSoakTime := T#0S;

FOR i := 1 TO 4 DO
	//Solvents and Times
	GVL_Recipe.stCurrentRecipe.stSolventsTimes.aSolventN[i] := 0;
	GVL_Recipe.stCurrentRecipe.stSolventsTimes.aTime[i] := T#0S;
	GVL_Recipe.stCurrentRecipe.stSolventsTimes.aVelocity[i] := 0;
	
	//Volumes
	GVL_Recipe.stCurrentRecipe.stVolumes.aF_Volume[i] := 0;
	GVL_Recipe.stCurrentRecipe.stVolumes.aS0_Volume[i] := 0;
	GVL_Recipe.stCurrentRecipe.stVolumes.aS1_Volume[i] := 0;
	GVL_Recipe.stCurrentRecipe.stVolumes.aS2_Volume[i] := 0;
	GVL_Recipe.stCurrentRecipe.stVolumes.aS3_Volume[i] := 0;
	GVL_Recipe.stCurrentRecipe.stVolumes.aS4_Volume[i] := 0;
	GVL_Recipe.stCurrentRecipe.stVolumes.aS5_Volume[i] := 0;
	GVL_Recipe.stCurrentRecipe.stVolumes.aS6_Volume[i] := 0;
	GVL_Recipe.stCurrentRecipe.stVolumes.aS7_Volume[i] := 0;
	GVL_Recipe.stCurrentRecipe.stVolumes.aT_IC_Volume[i] := 0;
END_FOR
END_ACTION

ACTION ACT_DatagridsRowNaming:
//Naming the HMI Recipe Screen Datagrid rows
//TcHmiDatagrid_SolventAndTimes
GVL_HMI.aSolventAndTimesRows[1].Parameter := 'Solvent #';
GVL_HMI.aSolventAndTimesRows[2].Parameter := 'Time';
GVL_HMI.aSolventAndTimesRows[3].Parameter := 'Velocity';

//TcHmiDatagrid_Volumes
GVL_HMI.aVolumeRows[1].Stage := 'T/IC';
GVL_HMI.aVolumeRows[2].Stage := 'S0';
GVL_HMI.aVolumeRows[3].Stage := 'S1';
GVL_HMI.aVolumeRows[4].Stage := 'S2';
GVL_HMI.aVolumeRows[5].Stage := 'S3';
GVL_HMI.aVolumeRows[6].Stage := 'S4';
GVL_HMI.aVolumeRows[7].Stage := 'S5';
GVL_HMI.aVolumeRows[8].Stage := 'S6';
GVL_HMI.aVolumeRows[9].Stage := 'S7';
GVL_HMI.aVolumeRows[10].Stage := 'F';

//TcHmiDatagrid_OtherParams
GVL_HMI.aOtherParamsRows[1].Parameter := 'Soak Time';
GVL_HMI.aOtherParamsRows[2].Parameter := 'Agitate 1 Time';
GVL_HMI.aOtherParamsRows[3].Parameter := 'Agitate 2 Time';
GVL_HMI.aOtherParamsRows[4].Parameter := 'Vials to Fill';
GVL_HMI.aOtherParamsRows[5].Parameter := 'Vial Prime Vol';
GVL_HMI.aOtherParamsRows[6].Parameter := 'Vial 1 Fill Vol';
GVL_HMI.aOtherParamsRows[7].Parameter := 'Vials 2-4 Fill Vol';
GVL_HMI.aOtherParamsRows[8].Parameter := 'Air Dry Time';
//TcHmiDatagrid_OtherParams - Data Units
GVL_HMI.aOtherParamsRows[1].Units     := 'sec';
GVL_HMI.aOtherParamsRows[2].Units     := 'sec';
GVL_HMI.aOtherParamsRows[3].Units     := 'sec';
GVL_HMI.aOtherParamsRows[4].Units     := 'unit';
GVL_HMI.aOtherParamsRows[5].Units     := 'ml';
GVL_HMI.aOtherParamsRows[6].Units     := 'ml';
GVL_HMI.aOtherParamsRows[7].Units     := 'ml';
GVL_HMI.aOtherParamsRows[8].Units     := 'sec';

//Finish the naming
bDatagridRowsNaming := TRUE;
END_ACTION

ACTION ACT_DatagridToRecipe:
IF NOT bDatagridToRecipeDone THEN
	// ---- Commit RecipeInfo ----	
	GVL_Recipe.stCurrentRecipe.stInfo.sCreatedBy := GVL_HMI.stRecipeInfo.sCreatedBy;
	GVL_Recipe.stCurrentRecipe.stInfo.sMethodName := GVL_HMI.stRecipeInfo.sMethodName;
	

	// ---- Commit SolventAndTimes ----
	FOR i := 1 TO 4 DO // 1: Rinse1, 2: Rinse2, 3: Wash1, 4: Wash2
		// Solvent #
		CASE i OF
			1: GVL_Recipe.stCurrentRecipe.stSolventsTimes.aSolventN[i] := TO_USINT(GVL_HMI.aSolventAndTimesRows[1].Rinse1);
			2: GVL_Recipe.stCurrentRecipe.stSolventsTimes.aSolventN[i] := TO_USINT(GVL_HMI.aSolventAndTimesRows[1].Rinse2);
			3: GVL_Recipe.stCurrentRecipe.stSolventsTimes.aSolventN[i] := TO_USINT(GVL_HMI.aSolventAndTimesRows[1].Wash1);
			4: GVL_Recipe.stCurrentRecipe.stSolventsTimes.aSolventN[i] := TO_USINT(GVL_HMI.aSolventAndTimesRows[1].Wash2);
		END_CASE;
		// Time (convertendo para TIME)
		CASE i OF
			1: GVL_Recipe.stCurrentRecipe.stSolventsTimes.aTime[i] := DWORD_TO_TIME(GVL_HMI.aSolventAndTimesRows[2].Rinse1 * 1000);
			2: GVL_Recipe.stCurrentRecipe.stSolventsTimes.aTime[i] := DWORD_TO_TIME(GVL_HMI.aSolventAndTimesRows[2].Rinse2 * 1000);
			3: GVL_Recipe.stCurrentRecipe.stSolventsTimes.aTime[i] := DWORD_TO_TIME(GVL_HMI.aSolventAndTimesRows[2].Wash1 * 1000);
			4: GVL_Recipe.stCurrentRecipe.stSolventsTimes.aTime[i] := DWORD_TO_TIME(GVL_HMI.aSolventAndTimesRows[2].Wash2 * 1000);
		END_CASE;
		// Velocity
		CASE i OF
			1: GVL_Recipe.stCurrentRecipe.stSolventsTimes.aVelocity[i] := GVL_HMI.aSolventAndTimesRows[3].Rinse1;
			2: GVL_Recipe.stCurrentRecipe.stSolventsTimes.aVelocity[i] := GVL_HMI.aSolventAndTimesRows[3].Rinse2;
			3: GVL_Recipe.stCurrentRecipe.stSolventsTimes.aVelocity[i] := GVL_HMI.aSolventAndTimesRows[3].Wash1;
			4: GVL_Recipe.stCurrentRecipe.stSolventsTimes.aVelocity[i] := GVL_HMI.aSolventAndTimesRows[3].Wash2;
		END_CASE;
	END_FOR
	
	// ---- Commit Volumes ----
	// Cada linha do aVolumesRows corresponde a um array do struct
	// Ordem: 1:T_IC, 2:S0, 3:S1, 4:S2, 5:S3, 6:S4, 7:S5, 8:S6, 9:S7, 10:F
	FOR i := 1 TO 4 DO // Rinse1, Rinse2, Wash1, Wash2
		// T_IC
		CASE i OF
			1: GVL_Recipe.stCurrentRecipe.stVolumes.aT_IC_Volume[i] := GVL_HMI.aVolumeRows[1].Rinse1;
			2: GVL_Recipe.stCurrentRecipe.stVolumes.aT_IC_Volume[i] := GVL_HMI.aVolumeRows[1].Rinse2;
			3: GVL_Recipe.stCurrentRecipe.stVolumes.aT_IC_Volume[i] := GVL_HMI.aVolumeRows[1].Wash1;
			4: GVL_Recipe.stCurrentRecipe.stVolumes.aT_IC_Volume[i] := GVL_HMI.aVolumeRows[1].Wash2;
		END_CASE;
		// S0
		CASE i OF
			1: GVL_Recipe.stCurrentRecipe.stVolumes.aS0_Volume[i] := GVL_HMI.aVolumeRows[2].Rinse1;
			2: GVL_Recipe.stCurrentRecipe.stVolumes.aS0_Volume[i] := GVL_HMI.aVolumeRows[2].Rinse2;
			3: GVL_Recipe.stCurrentRecipe.stVolumes.aS0_Volume[i] := GVL_HMI.aVolumeRows[2].Wash1;
			4: GVL_Recipe.stCurrentRecipe.stVolumes.aS0_Volume[i] := GVL_HMI.aVolumeRows[2].Wash2;
		END_CASE;
		// S1 
		CASE i OF
			1: GVL_Recipe.stCurrentRecipe.stVolumes.aS1_Volume[i] := GVL_HMI.aVolumeRows[3].Rinse1;
			2: GVL_Recipe.stCurrentRecipe.stVolumes.aS1_Volume[i] := GVL_HMI.aVolumeRows[3].Rinse2;
			3: GVL_Recipe.stCurrentRecipe.stVolumes.aS1_Volume[i] := GVL_HMI.aVolumeRows[3].Wash1;
			4: GVL_Recipe.stCurrentRecipe.stVolumes.aS1_Volume[i] := GVL_HMI.aVolumeRows[3].Wash2;
		END_CASE;
		// S2
		CASE i OF
			1: GVL_Recipe.stCurrentRecipe.stVolumes.aS2_Volume[i] := GVL_HMI.aVolumeRows[4].Rinse1;
			2: GVL_Recipe.stCurrentRecipe.stVolumes.aS2_Volume[i] := GVL_HMI.aVolumeRows[4].Rinse2;
			3: GVL_Recipe.stCurrentRecipe.stVolumes.aS2_Volume[i] := GVL_HMI.aVolumeRows[4].Wash1;
			4: GVL_Recipe.stCurrentRecipe.stVolumes.aS2_Volume[i] := GVL_HMI.aVolumeRows[4].Wash2;
		END_CASE;
		CASE i OF
			1: GVL_Recipe.stCurrentRecipe.stVolumes.aS3_Volume[i] := GVL_HMI.aVolumeRows[5].Rinse1;
			2: GVL_Recipe.stCurrentRecipe.stVolumes.aS3_Volume[i] := GVL_HMI.aVolumeRows[5].Rinse2;
			3: GVL_Recipe.stCurrentRecipe.stVolumes.aS3_Volume[i] := GVL_HMI.aVolumeRows[5].Wash1;
			4: GVL_Recipe.stCurrentRecipe.stVolumes.aS3_Volume[i] := GVL_HMI.aVolumeRows[5].Wash2;
		END_CASE;
		CASE i OF
			1: GVL_Recipe.stCurrentRecipe.stVolumes.aS4_Volume[i] := GVL_HMI.aVolumeRows[6].Rinse1;
			2: GVL_Recipe.stCurrentRecipe.stVolumes.aS4_Volume[i] := GVL_HMI.aVolumeRows[6].Rinse2;
			3: GVL_Recipe.stCurrentRecipe.stVolumes.aS4_Volume[i] := GVL_HMI.aVolumeRows[6].Wash1;
			4: GVL_Recipe.stCurrentRecipe.stVolumes.aS4_Volume[i] := GVL_HMI.aVolumeRows[6].Wash2;
		END_CASE;
		CASE i OF
			1: GVL_Recipe.stCurrentRecipe.stVolumes.aS5_Volume[i] := GVL_HMI.aVolumeRows[7].Rinse1;
			2: GVL_Recipe.stCurrentRecipe.stVolumes.aS5_Volume[i] := GVL_HMI.aVolumeRows[7].Rinse2;
			3: GVL_Recipe.stCurrentRecipe.stVolumes.aS5_Volume[i] := GVL_HMI.aVolumeRows[7].Wash1;
			4: GVL_Recipe.stCurrentRecipe.stVolumes.aS5_Volume[i] := GVL_HMI.aVolumeRows[7].Wash2;
		END_CASE;
		CASE i OF
			1: GVL_Recipe.stCurrentRecipe.stVolumes.aS6_Volume[i] := GVL_HMI.aVolumeRows[8].Rinse1;
			2: GVL_Recipe.stCurrentRecipe.stVolumes.aS6_Volume[i] := GVL_HMI.aVolumeRows[8].Rinse2;
			3: GVL_Recipe.stCurrentRecipe.stVolumes.aS6_Volume[i] := GVL_HMI.aVolumeRows[8].Wash1;
			4: GVL_Recipe.stCurrentRecipe.stVolumes.aS6_Volume[i] := GVL_HMI.aVolumeRows[8].Wash2;
		END_CASE;
		CASE i OF
			1: GVL_Recipe.stCurrentRecipe.stVolumes.aS7_Volume[i] := GVL_HMI.aVolumeRows[9].Rinse1;
			2: GVL_Recipe.stCurrentRecipe.stVolumes.aS7_Volume[i] := GVL_HMI.aVolumeRows[9].Rinse2;
			3: GVL_Recipe.stCurrentRecipe.stVolumes.aS7_Volume[i] := GVL_HMI.aVolumeRows[9].Wash1;
			4: GVL_Recipe.stCurrentRecipe.stVolumes.aS7_Volume[i] := GVL_HMI.aVolumeRows[9].Wash2;
		END_CASE;
		CASE i OF
			1: GVL_Recipe.stCurrentRecipe.stVolumes.aF_Volume[i] := GVL_HMI.aVolumeRows[10].Rinse1;
			2: GVL_Recipe.stCurrentRecipe.stVolumes.aF_Volume[i] := GVL_HMI.aVolumeRows[10].Rinse2;
			3: GVL_Recipe.stCurrentRecipe.stVolumes.aF_Volume[i] := GVL_HMI.aVolumeRows[10].Wash1;
			4: GVL_Recipe.stCurrentRecipe.stVolumes.aF_Volume[i] := GVL_HMI.aVolumeRows[10].Wash2;
		END_CASE;
	END_FOR
	
	// ---- Commit OtherParams ----
	// Supondo a ordem das linhas conforme DataGrid (ajuste se necessário)
	GVL_Recipe.stCurrentRecipe.stOtherParams.tSoakTime        := TO_TIME(GVL_HMI.aOtherParamsRows[1].Value * 1000);
	GVL_Recipe.stCurrentRecipe.stOtherParams.tAgitate1Time    := TO_TIME(GVL_HMI.aOtherParamsRows[2].Value * 1000);
	GVL_Recipe.stCurrentRecipe.stOtherParams.tAgitate2Time    := TO_TIME(GVL_HMI.aOtherParamsRows[3].Value * 1000);
	GVL_Recipe.stCurrentRecipe.stOtherParams.iVialsToFill     := TO_USINT(GVL_HMI.aOtherParamsRows[4].Value);
	GVL_Recipe.stCurrentRecipe.stOtherParams.rVialPrimeVol    := GVL_HMI.aOtherParamsRows[5].Value;
	GVL_Recipe.stCurrentRecipe.stOtherParams.rVial1FillVol    := GVL_HMI.aOtherParamsRows[6].Value;
	GVL_Recipe.stCurrentRecipe.stOtherParams.rVials2_4FillVol := GVL_HMI.aOtherParamsRows[7].Value;
	GVL_Recipe.stCurrentRecipe.stOtherParams.tAirDryTime   	  := TO_TIME(GVL_HMI.aOtherParamsRows[8].Value * 1000);
	
	//reset flags
	
	i:=0;
	
	DB_Edit_Method(start:=TRUE);
	
	
END_IF
END_ACTION

ACTION ACT_PopulateDeleteRecipeInfo:
// Fill up the info fields for popup delete confirmation
GVL_HMI.stDeleteRecipeInfo.sCreatedBy := GVL_Recipe.stCurrentRecipe.stInfo.sCreatedBy;
GVL_HMI.stDeleteRecipeInfo.dCreationDate := GVL_Recipe.stCurrentRecipe.stInfo.dCreationDate;
GVL_HMI.stDeleteRecipeInfo.iRevision := GVL_Recipe.stCurrentRecipe.stInfo.iRevision;
GVL_HMI.stDeleteRecipeInfo.sMethodName := GVL_Recipe.stCurrentRecipe.stInfo.sMethodName;
GVL_HMI.stDeleteRecipeInfo.sFileName := GVL_Recipe.sSelectedRecipeName;

// Resets the flag
GVL_HMI.bDeleteRecipeButton := FALSE;
END_ACTION

ACTION ACT_RecipeToDatagrid:

// SolventAndTimes
GVL_HMI.aSolventAndTimesRows[1].Rinse1 := GVL_Recipe.stCurrentRecipe.stSolventsTimes.aSolventN[1];
GVL_HMI.aSolventAndTimesRows[1].Rinse2 := GVL_Recipe.stCurrentRecipe.stSolventsTimes.aSolventN[2];
GVL_HMI.aSolventAndTimesRows[1].Wash1  := GVL_Recipe.stCurrentRecipe.stSolventsTimes.aSolventN[3];
GVL_HMI.aSolventAndTimesRows[1].Wash2  := GVL_Recipe.stCurrentRecipe.stSolventsTimes.aSolventN[4];

GVL_HMI.aSolventAndTimesRows[2].Rinse1 := TO_INT(TIME_TO_DWORD(GVL_Recipe.stCurrentRecipe.stSolventsTimes.aTime[1])/1000);
GVL_HMI.aSolventAndTimesRows[2].Rinse2 := TO_INT(TIME_TO_DWORD(GVL_Recipe.stCurrentRecipe.stSolventsTimes.aTime[2])/1000);
GVL_HMI.aSolventAndTimesRows[2].Wash1  := TO_INT(TIME_TO_DWORD(GVL_Recipe.stCurrentRecipe.stSolventsTimes.aTime[3])/1000);
GVL_HMI.aSolventAndTimesRows[2].Wash2  := TO_INT(TIME_TO_DWORD(GVL_Recipe.stCurrentRecipe.stSolventsTimes.aTime[4])/1000);

GVL_HMI.aSolventAndTimesRows[3].Rinse1 := GVL_Recipe.stCurrentRecipe.stSolventsTimes.aVelocity[1];
GVL_HMI.aSolventAndTimesRows[3].Rinse2 := GVL_Recipe.stCurrentRecipe.stSolventsTimes.aVelocity[2];
GVL_HMI.aSolventAndTimesRows[3].Wash1  := GVL_Recipe.stCurrentRecipe.stSolventsTimes.aVelocity[3];
GVL_HMI.aSolventAndTimesRows[3].Wash2  := GVL_Recipe.stCurrentRecipe.stSolventsTimes.aVelocity[4];

// Volumes
GVL_HMI.aVolumeRows[1].Rinse1 := GVL_Recipe.stCurrentRecipe.stVolumes.aT_IC_Volume[1];
GVL_HMI.aVolumeRows[1].Rinse2 := GVL_Recipe.stCurrentRecipe.stVolumes.aT_IC_Volume[2];
GVL_HMI.aVolumeRows[1].Wash1  := GVL_Recipe.stCurrentRecipe.stVolumes.aT_IC_Volume[3];
GVL_HMI.aVolumeRows[1].Wash2  := GVL_Recipe.stCurrentRecipe.stVolumes.aT_IC_Volume[4];

GVL_HMI.aVolumeRows[2].Rinse1 := GVL_Recipe.stCurrentRecipe.stVolumes.aS0_Volume[1];
GVL_HMI.aVolumeRows[2].Rinse2 := GVL_Recipe.stCurrentRecipe.stVolumes.aS0_Volume[2];
GVL_HMI.aVolumeRows[2].Wash1  := GVL_Recipe.stCurrentRecipe.stVolumes.aS0_Volume[3];
GVL_HMI.aVolumeRows[2].Wash2  := GVL_Recipe.stCurrentRecipe.stVolumes.aS0_Volume[4];

GVL_HMI.aVolumeRows[3].Rinse1 := GVL_Recipe.stCurrentRecipe.stVolumes.aS1_Volume[1];
GVL_HMI.aVolumeRows[3].Rinse2 := GVL_Recipe.stCurrentRecipe.stVolumes.aS1_Volume[2];
GVL_HMI.aVolumeRows[3].Wash1  := GVL_Recipe.stCurrentRecipe.stVolumes.aS1_Volume[3];
GVL_HMI.aVolumeRows[3].Wash2  := GVL_Recipe.stCurrentRecipe.stVolumes.aS1_Volume[4];

GVL_HMI.aVolumeRows[4].Rinse1 := GVL_Recipe.stCurrentRecipe.stVolumes.aS2_Volume[1];
GVL_HMI.aVolumeRows[4].Rinse2 := GVL_Recipe.stCurrentRecipe.stVolumes.aS2_Volume[2];
GVL_HMI.aVolumeRows[4].Wash1  := GVL_Recipe.stCurrentRecipe.stVolumes.aS2_Volume[3];
GVL_HMI.aVolumeRows[4].Wash2  := GVL_Recipe.stCurrentRecipe.stVolumes.aS2_Volume[4];

GVL_HMI.aVolumeRows[5].Rinse1 := GVL_Recipe.stCurrentRecipe.stVolumes.aS3_Volume[1];
GVL_HMI.aVolumeRows[5].Rinse2 := GVL_Recipe.stCurrentRecipe.stVolumes.aS3_Volume[2];
GVL_HMI.aVolumeRows[5].Wash1  := GVL_Recipe.stCurrentRecipe.stVolumes.aS3_Volume[3];
GVL_HMI.aVolumeRows[5].Wash2  := GVL_Recipe.stCurrentRecipe.stVolumes.aS3_Volume[4];

GVL_HMI.aVolumeRows[6].Rinse1 := GVL_Recipe.stCurrentRecipe.stVolumes.aS4_Volume[1];
GVL_HMI.aVolumeRows[6].Rinse2 := GVL_Recipe.stCurrentRecipe.stVolumes.aS4_Volume[2];
GVL_HMI.aVolumeRows[6].Wash1  := GVL_Recipe.stCurrentRecipe.stVolumes.aS4_Volume[3];
GVL_HMI.aVolumeRows[6].Wash2  := GVL_Recipe.stCurrentRecipe.stVolumes.aS4_Volume[4];

GVL_HMI.aVolumeRows[7].Rinse1 := GVL_Recipe.stCurrentRecipe.stVolumes.aS5_Volume[1];
GVL_HMI.aVolumeRows[7].Rinse2 := GVL_Recipe.stCurrentRecipe.stVolumes.aS5_Volume[2];
GVL_HMI.aVolumeRows[7].Wash1  := GVL_Recipe.stCurrentRecipe.stVolumes.aS5_Volume[3];
GVL_HMI.aVolumeRows[7].Wash2  := GVL_Recipe.stCurrentRecipe.stVolumes.aS5_Volume[4];

GVL_HMI.aVolumeRows[8].Rinse1 := GVL_Recipe.stCurrentRecipe.stVolumes.aS6_Volume[1];
GVL_HMI.aVolumeRows[8].Rinse2 := GVL_Recipe.stCurrentRecipe.stVolumes.aS6_Volume[2];
GVL_HMI.aVolumeRows[8].Wash1  := GVL_Recipe.stCurrentRecipe.stVolumes.aS6_Volume[3];
GVL_HMI.aVolumeRows[8].Wash2  := GVL_Recipe.stCurrentRecipe.stVolumes.aS6_Volume[4];

GVL_HMI.aVolumeRows[9].Rinse1 := GVL_Recipe.stCurrentRecipe.stVolumes.aS7_Volume[1];
GVL_HMI.aVolumeRows[9].Rinse2 := GVL_Recipe.stCurrentRecipe.stVolumes.aS7_Volume[2];
GVL_HMI.aVolumeRows[9].Wash1  := GVL_Recipe.stCurrentRecipe.stVolumes.aS7_Volume[3];
GVL_HMI.aVolumeRows[9].Wash2  := GVL_Recipe.stCurrentRecipe.stVolumes.aS7_Volume[4];

GVL_HMI.aVolumeRows[10].Rinse1 := GVL_Recipe.stCurrentRecipe.stVolumes.aF_Volume[1];
GVL_HMI.aVolumeRows[10].Rinse2 := GVL_Recipe.stCurrentRecipe.stVolumes.aF_Volume[2];
GVL_HMI.aVolumeRows[10].Wash1  := GVL_Recipe.stCurrentRecipe.stVolumes.aF_Volume[3];
GVL_HMI.aVolumeRows[10].Wash2  := GVL_Recipe.stCurrentRecipe.stVolumes.aF_Volume[4];

// --- Outros Params ---
GVL_HMI.aOtherParamsRows[1].Value := UDINT_TO_REAL(TIME_TO_DWORD(GVL_Recipe.stCurrentRecipe.stOtherParams.tSoakTime)/1000);
GVL_HMI.aOtherParamsRows[2].Value := UDINT_TO_REAL(TIME_TO_DWORD(GVL_Recipe.stCurrentRecipe.stOtherParams.tAgitate1Time)/1000);
GVL_HMI.aOtherParamsRows[3].Value := UDINT_TO_REAL(TIME_TO_DWORD(GVL_Recipe.stCurrentRecipe.stOtherParams.tAgitate2Time)/1000);
GVL_HMI.aOtherParamsRows[4].Value := GVL_Recipe.stCurrentRecipe.stOtherParams.iVialsToFill;
GVL_HMI.aOtherParamsRows[5].Value := GVL_Recipe.stCurrentRecipe.stOtherParams.rVialPrimeVol;
GVL_HMI.aOtherParamsRows[6].Value := GVL_Recipe.stCurrentRecipe.stOtherParams.rVial1FillVol;
GVL_HMI.aOtherParamsRows[7].Value := GVL_Recipe.stCurrentRecipe.stOtherParams.rVials2_4FillVol;
GVL_HMI.aOtherParamsRows[8].Value := UDINT_TO_REAL(TIME_TO_DWORD(GVL_Recipe.stCurrentRecipe.stOtherParams.tAirDryTime)/1000);

//Flag to initiate the save fb
GVL_HMI.bReloadRecipeDatagrids  := FALSE;
END_ACTION

END_PROGRAM

// ---- POUs/4. RecipeHandle/FB_LoadRecipe.TcPOU
FUNCTION_BLOCK FB_LoadRecipe
VAR_INPUT
	sFileName : STRING(255); // Ex: 'C:\TwinCAT\Recipes\NomeDaReceita.json'
    bExecute  : BOOL;
END_VAR
VAR_OUTPUT
	bBusy   : BOOL;
    bDone   : BOOL;
    bError  : BOOL;
    nErrId  : UDINT;
END_VAR
VAR
	fbFileOpen  : FB_FileOpen;
    fbFileRead  : FB_FileRead;
    fbFileClose : FB_FileClose;
    fbJson      : FB_JsonDomParser;

    hFile    	: UINT;
    sBuffer  	: STRING(16384);
    jsonRoot 	: SJsonValue;
    jsonVal  	: SJsonValue;
	nBytesRead  : UDINT;
    idx      	: INT;
    iStep     	: INT;

    sPath    : STRING(255);
END_VAR

IF NOT bExecute THEN
	bBusy := FALSE;
	bDone := FALSE;
	bError := FALSE;
	nErrId := 0;
	sBuffer := '';
	fbFileOpen(bExecute := FALSE);
	fbFileRead(bExecute := FALSE);
	fbFileClose(bExecute := FALSE);
	iStep := 0;
END_IF


CASE iStep OF
0:
    IF bExecute THEN
        bBusy := TRUE;
        bDone := FALSE;
        bError := FALSE;
        nErrId := 0;

        fbFileOpen(
            sNetId := '',
            sPathName := sFileName,
            nMode := FOPEN_MODEREAD OR FOPEN_MODETEXT,
            bExecute := TRUE
        );
		sBuffer := '';
        iStep := 10;
    END_IF

10:
    fbFileOpen(bExecute := FALSE);
    IF NOT fbFileOpen.bBusy THEN
        IF fbFileOpen.bError THEN
            bError := TRUE;
            nErrId := fbFileOpen.nErrId;
            iStep := 100;
        ELSE
            hFile := fbFileOpen.hFile;
            fbFileRead(
                sNetId := '',
                hFile := hFile,
                pReadBuff := ADR(sBuffer),
                cbReadLen := SIZEOF(sBuffer),
                bExecute := TRUE
            );
            iStep := 20;
        END_IF
    END_IF

20:
    fbFileRead(bExecute := FALSE, sNetId := '', hFile := hFile, pReadBuff := ADR(sBuffer), cbReadLen := SIZEOF(sBuffer), cbRead => nBytesRead);
    IF NOT fbFileRead.bBusy THEN
        IF fbFileRead.bError THEN
            bError := TRUE;
            nErrId := fbFileRead.nErrId;
            iStep := 90;
        ELSE
			// Clear the buffer
            IF nBytesRead < SIZEOF(sBuffer) THEN
    			sBuffer[nBytesRead] := 0; 
			END_IF
            fbFileClose(sNetId := '', hFile := hFile, bExecute := TRUE);
            iStep := 30;
        END_IF
    END_IF

30:
    fbFileClose(bExecute := FALSE);
    IF NOT fbFileClose.bBusy THEN
        IF fbFileClose.bError THEN
            bError := TRUE;
            nErrId := fbFileClose.nErrId;
            iStep := 100;
        ELSE
            iStep := 40;
        END_IF
    END_IF

40:
    jsonRoot := fbJson.ParseDocument(sBuffer);
    IF jsonRoot = 0 THEN
        bError := TRUE;
        nErrId := 16#F1000001; // Código customizado para JSON inválido
        iStep := 100;
    ELSE
        iStep := 50;
    END_IF

50: //Fill the variables with Json buffer info [Parse Json file]
    sPath := 'stInfo/sMethodName';
    GVL_Recipe.stCurrentRecipe.stInfo.sMethodName := fbJson.GetString(fbJson.FindMemberPath(jsonRoot, sPath));

    sPath := 'stInfo/sCreatedBy';
    GVL_Recipe.stCurrentRecipe.stInfo.sCreatedBy := fbJson.GetString(fbJson.FindMemberPath(jsonRoot, sPath));

    sPath := 'stInfo/dCreationDate';
    GVL_Recipe.stCurrentRecipe.stInfo.dCreationDate := STRING_TO_DATE(fbJson.GetString(fbJson.FindMemberPath(jsonRoot, sPath)));

    sPath := 'stInfo/iRevision';
    GVL_Recipe.stCurrentRecipe.stInfo.iRevision := DINT_TO_INT(fbJson.GetInt(fbJson.FindMemberPath(jsonRoot, sPath)));

    FOR idx := 1 TO 4 DO
        sPath := CONCAT('stSolventsTimes/aSolventN#', INT_TO_STRING(idx-1));
        GVL_Recipe.stCurrentRecipe.stSolventsTimes.aSolventN[idx] := TO_USINT(fbJson.GetInt(fbJson.FindMemberPath(jsonRoot, sPath)));

        sPath := CONCAT('stSolventsTimes/aTime#', INT_TO_STRING(idx-1));
        GVL_Recipe.stCurrentRecipe.stSolventsTimes.aTime[idx] := STRING_TO_TIME(fbJson.GetString(fbJson.FindMemberPath(jsonRoot, sPath)));

        sPath := CONCAT('stSolventsTimes/aVelocity#', INT_TO_STRING(idx-1));
        GVL_Recipe.stCurrentRecipe.stSolventsTimes.aVelocity[idx] := TO_INT(fbJson.GetInt(fbJson.FindMemberPath(jsonRoot, sPath)));
    END_FOR

    FOR idx := 1 TO 4 DO
        sPath := CONCAT('stVolumes/aT_IC_Volume#', INT_TO_STRING(idx-1));
        GVL_Recipe.stCurrentRecipe.stVolumes.aT_IC_Volume[idx] := LREAL_TO_REAL(fbJson.GetDouble(fbJson.FindMemberPath(jsonRoot, sPath)));
		
		sPath := CONCAT('stVolumes/aS0_Volume#', INT_TO_STRING(idx-1));
        GVL_Recipe.stCurrentRecipe.stVolumes.aS0_Volume[idx] := LREAL_TO_REAL(fbJson.GetDouble(fbJson.FindMemberPath(jsonRoot, sPath)));
		
		sPath := CONCAT('stVolumes/aS1_Volume#', INT_TO_STRING(idx-1));
        GVL_Recipe.stCurrentRecipe.stVolumes.aS1_Volume[idx] := LREAL_TO_REAL(fbJson.GetDouble(fbJson.FindMemberPath(jsonRoot, sPath)));
		
		sPath := CONCAT('stVolumes/aS2_Volume#', INT_TO_STRING(idx-1));
        GVL_Recipe.stCurrentRecipe.stVolumes.aS2_Volume[idx] := LREAL_TO_REAL(fbJson.GetDouble(fbJson.FindMemberPath(jsonRoot, sPath)));
		
		sPath := CONCAT('stVolumes/aS3_Volume#', INT_TO_STRING(idx-1));
        GVL_Recipe.stCurrentRecipe.stVolumes.aS3_Volume[idx] := LREAL_TO_REAL(fbJson.GetDouble(fbJson.FindMemberPath(jsonRoot, sPath)));
		
		sPath := CONCAT('stVolumes/aS4_Volume#', INT_TO_STRING(idx-1));
        GVL_Recipe.stCurrentRecipe.stVolumes.aS4_Volume[idx] := LREAL_TO_REAL(fbJson.GetDouble(fbJson.FindMemberPath(jsonRoot, sPath)));
		
		sPath := CONCAT('stVolumes/aS5_Volume#', INT_TO_STRING(idx-1));
        GVL_Recipe.stCurrentRecipe.stVolumes.aS5_Volume[idx] := LREAL_TO_REAL(fbJson.GetDouble(fbJson.FindMemberPath(jsonRoot, sPath)));
		
		sPath := CONCAT('stVolumes/aS6_Volume#', INT_TO_STRING(idx-1));
        GVL_Recipe.stCurrentRecipe.stVolumes.aS6_Volume[idx] := LREAL_TO_REAL(fbJson.GetDouble(fbJson.FindMemberPath(jsonRoot, sPath)));
		
		sPath := CONCAT('stVolumes/aS7_Volume#', INT_TO_STRING(idx-1));
        GVL_Recipe.stCurrentRecipe.stVolumes.aS7_Volume[idx] := LREAL_TO_REAL(fbJson.GetDouble(fbJson.FindMemberPath(jsonRoot, sPath)));
		
		sPath := CONCAT('stVolumes/aF_Volume#', INT_TO_STRING(idx-1));
        GVL_Recipe.stCurrentRecipe.stVolumes.aF_Volume[idx] := LREAL_TO_REAL(fbJson.GetDouble(fbJson.FindMemberPath(jsonRoot, sPath)));
		
    END_FOR

    sPath := 'stOtherParams/tSoakTime';
    GVL_Recipe.stCurrentRecipe.stOtherParams.tSoakTime := STRING_TO_TIME(fbJson.GetString(fbJson.FindMemberPath(jsonRoot, sPath)));
	
	sPath := 'stOtherParams/tAgitate1Time';
    GVL_Recipe.stCurrentRecipe.stOtherParams.tAgitate1Time := STRING_TO_TIME(fbJson.GetString(fbJson.FindMemberPath(jsonRoot, sPath)));
	
	sPath := 'stOtherParams/tAgitate2Time';
    GVL_Recipe.stCurrentRecipe.stOtherParams.tAgitate2Time := STRING_TO_TIME(fbJson.GetString(fbJson.FindMemberPath(jsonRoot, sPath)));
	
	sPath := 'stOtherParams/iVialsToFill';
    GVL_Recipe.stCurrentRecipe.stOtherParams.iVialsToFill := TO_USINT(fbJson.GetInt(fbJson.FindMemberPath(jsonRoot, sPath)));
	
	sPath := 'stOtherParams/rVialPrimeVol';
    GVL_Recipe.stCurrentRecipe.stOtherParams.rVialPrimeVol := LREAL_TO_REAL(fbJson.GetDouble(fbJson.FindMemberPath(jsonRoot, sPath)));
	
	sPath := 'stOtherParams/rVial1FillVol';
    GVL_Recipe.stCurrentRecipe.stOtherParams.rVial1FillVol := LREAL_TO_REAL(fbJson.GetDouble(fbJson.FindMemberPath(jsonRoot, sPath)));
	
	sPath := 'stOtherParams/rVials2_4FillVol';
    GVL_Recipe.stCurrentRecipe.stOtherParams.rVials2_4FillVol := LREAL_TO_REAL(fbJson.GetDouble(fbJson.FindMemberPath(jsonRoot, sPath)));
	
	sPath := 'stOtherParams/tAirDryTime';
    GVL_Recipe.stCurrentRecipe.stOtherParams.tAirDryTime := STRING_TO_TIME(fbJson.GetString(fbJson.FindMemberPath(jsonRoot, sPath)));

    iStep := 60;
	
60: // Fill the HMI datagrids for recipe screen
	//Recipe Header info
	GVL_HMI.stRecipeInfo.sMethodName := GVL_Recipe.stCurrentRecipe.stInfo.sMethodName;
	GVL_HMI.stRecipeInfo.sCreatedBy := GVL_Recipe.stCurrentRecipe.stInfo.sCreatedBy;
	GVL_HMI.stRecipeInfo.dCreationDate := GVL_Recipe.stCurrentRecipe.stInfo.dCreationDate;
	GVL_HMI.stRecipeInfo.iRevision := GVL_Recipe.stCurrentRecipe.stInfo.iRevision;
	
	// Solvents and Times datagrid
	// Row 1: Solvent #
	GVL_HMI.aSolventAndTimesRows[1].Rinse1 := GVL_Recipe.stCurrentRecipe.stSolventsTimes.aSolventN[1];
	GVL_HMI.aSolventAndTimesRows[1].Rinse2 := GVL_Recipe.stCurrentRecipe.stSolventsTimes.aSolventN[2];
	GVL_HMI.aSolventAndTimesRows[1].Wash1  := GVL_Recipe.stCurrentRecipe.stSolventsTimes.aSolventN[3];
	GVL_HMI.aSolventAndTimesRows[1].Wash2  := GVL_Recipe.stCurrentRecipe.stSolventsTimes.aSolventN[4];
	
